REGION Network 4: Current revision and modification history
   // ▄▄▄▄▄▄▄▄▄▄▄▄▄▄▄▄▄▄▄▄▄▄▄▄▄▄▄▄▄▄▄▄▄▄▄▄▄▄▄▄▄▄▄▄
   // MODIFICATION HISTORY
   // 
   // 
   // The revision data shown here, in the network comments, contains additional information 
   // reflecting the software development workflow under the version control system (VCS) employed 
   // to track all software changes.
   // 
   // The VCS in use is the Git Source Code Management system in conjunction with the GitHub online 
   // hosting system. The software in its entirety is available in the GitHub remote repository:
   // 
   //      https://github.com/practicalseries/PS2001-pal-software
   // 
   // The repository is public and can be freely copied (forked in GitHub terminology) and used 
   // under the MIT licence. 
   // 
   // The MIT licence is reproduced in full in the last network of this software module.
   // 
   // 
   //  ―――――――――――――――――――――――――――――――――――――――――――
   //  DATE       REVISION             MASTER BRANCH     DEV
   //          (nnn.amm)   COMMIT TAG    (Base ---> Merge)    BRANCH   Author
   //  ———————————————————————————————————————————
   //  2024.05.11    002.801   D0017A-000.104   D0017 N/A     D017A   M. Gledhill
   //                        RAW_ANALOG changed to AI_RAW_SIGNAL
   //                        AI_RAW_DATA and AI_SCALE_DATA added and
   //                        copied to DYNAMIC_DATA (see db00801 SMDS)
   // 
   //  2022.04.16    002.000   D0011      D0010 D0011  None  M. Gledhill
   //                        FC02001 — RELEASED FOR USE
   //                          Merge back to master branch
   // 
   //  2022.04.11    001.801   D0010A-000.801   D0010 N/A     D010A   M. Gledhill
   //                        Released for test (SCV)
   //  2022.04.08    001.102   D0010A-000.104   D0010 N/A     D010A   M. Gledhill
   //                        Temporary variable name change (cal)
   // 
   //  2022.04.05    001.101   D0010A-000.103   D0010 N/A     D010A   M. Gledhill
   //                        Over and under range based on scaled signal
   //                        INFO_TYPE, cal_OR_Abs and cal_UR_Abs added
   //                        Comments updated and standardised
   //                        UDT variable names standardised
   // 
   //  2021.05.26    001.000   D0008      D0006 D0008  None    M. Gledhill
   //                        FC02001 — RELEASED FOR USE
   //                          Merge back to master branch
   // 
   //  2021.05.26    001.000   D0006B-001.000   D0006 N/A     D0006B   M. Gledhill
   //                        FC02001 — Post-test RELEASED FOR USE
   // 
   //  2021.05.24    000.801   D0006B-000.801   D0006 N/A     D0006B   M. Gledhill
   //                        FC02001 — Released for SMT
   // 
   //  2021.05.18    000.101   D0006B-000.101   D0006 N/A     D0006B   M. Gledhill
   //                        FC02001 Migration to VCS
   //  ———————————————————————————————————————————
   //   Where: nnn  =  Major revision
   //         a  =  Type (1-7 Development, 8 Proving, 9 Qualification, 0 Release)
   //       mm  =  Minor revision (must be 00 if a = 0)
   //         Block properties version number should be set to nn.a (only one decimal place)
   // 
   // ▄▄▄▄▄▄▄▄▄▄▄▄▄▄▄▄▄▄▄▄▄▄▄▄▄▄▄▄▄▄▄▄▄▄▄▄▄▄▄▄▄▄▄▄
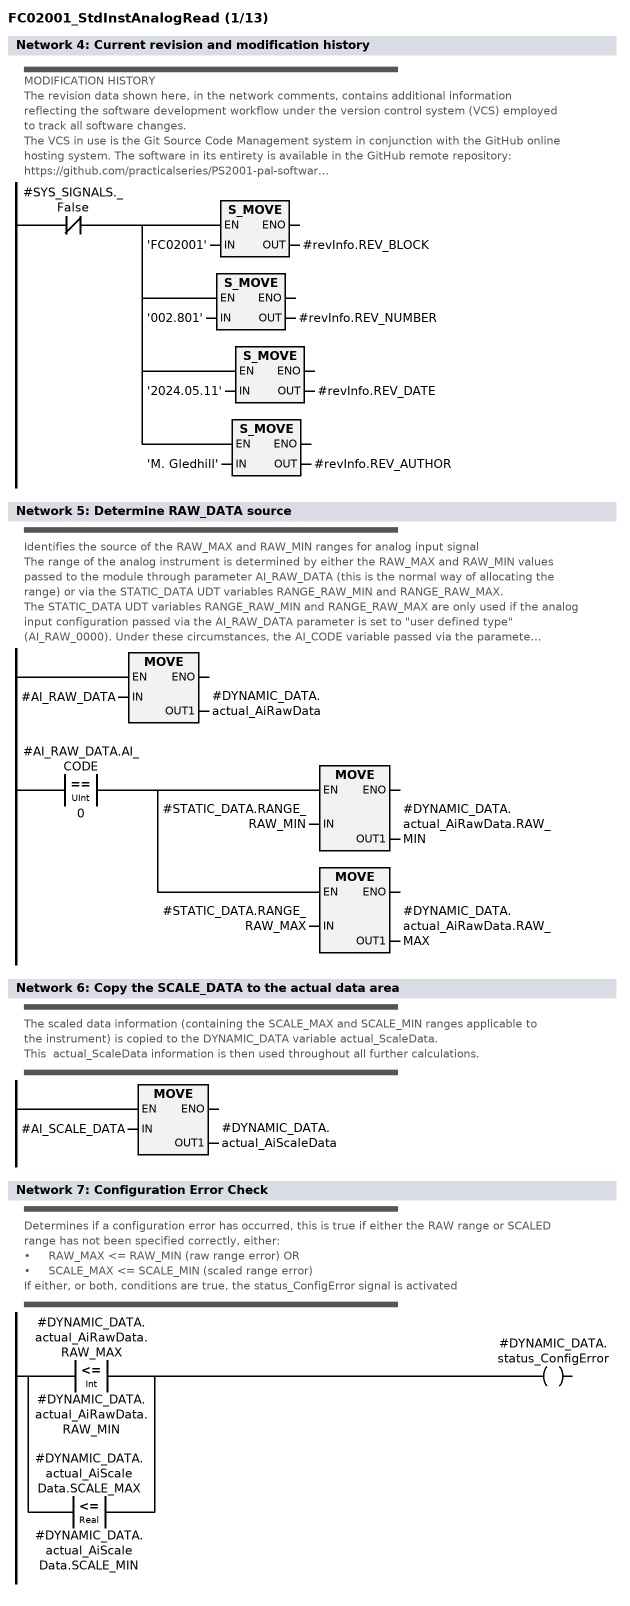
   RUNG wire#powerrail
      I_Contact( #SYS_SIGNALS._False )
      wire#w1
      S_Move(in := 'FC02001', out => #revInfo.REV_BLOCK)
   END_RUNG
   RUNG wire#w1
      S_Move(in := '002.801', out => #revInfo.REV_NUMBER)
   END_RUNG
   RUNG wire#w1
      S_Move(in := '2024.05.11', out => #revInfo.REV_DATE)
   END_RUNG
   RUNG wire#w1
      S_Move(in := 'M. Gledhill', out => #revInfo.REV_AUTHOR)
   END_RUNG
   // the same network as SCL:
   IF NOT #SYS_SIGNALS._False THEN
       #revInfo.REV_BLOCK := 'FC02001';
       #revInfo.REV_NUMBER := '002.801';
       #revInfo.REV_DATE := '2024.05.11';
       #revInfo.REV_AUTHOR := 'M. Gledhill';
   END_IF;
END_REGION

REGION Network 5: Determine RAW_DATA source
   // ▀▀▀▀▀▀▀▀▀▀▀▀▀▀▀▀▀▀▀▀▀▀▀▀▀▀▀▀▀▀▀▀▀▀▀▀▀▀▀▀▀▀▀▀
   // Identifies the source of the RAW_MAX and RAW_MIN ranges for analog input signal
   // 
   // The range of the analog instrument is determined by either the RAW_MAX and RAW_MIN values 
   // passed to the module through parameter AI_RAW_DATA (this is the normal way of allocating the 
   // range) or via the STATIC_DATA UDT variables RANGE_RAW_MIN and RANGE_RAW_MAX.
   // 
   // 
   // The STATIC_DATA UDT variables RANGE_RAW_MIN and RANGE_RAW_MAX are only used if the analog
   // input configuration passed via the AI_RAW_DATA parameter is set to "user defined type" 
   // (AI_RAW_0000). Under these circumstances, the AI_CODE variable passed via the parameter 
   // AI_RAW_DATA will be set to zero and the STATIC_DATA UDT variables RANGE_RAW_MIN and 
   // RANGE_RAW_MAX are to be used in place of the range data given via the AI_RAW_DATA parameter.
   // 
   // Irrespective of the source, the RAW_MIN and RAW_MAX data in use will be copied to the 
   // DYNAMIC_DATA variable actual_RawData.
   // ▄▄▄▄▄▄▄▄▄▄▄▄▄▄▄▄▄▄▄▄▄▄▄▄▄▄▄▄▄▄▄▄▄▄▄▄▄▄▄▄▄▄▄▄
   RUNG wire#powerrail
      Move(in := #AI_RAW_DATA, out1 => #DYNAMIC_DATA.actual_AiRawData)
   END_RUNG
   RUNG wire#powerrail
      { S7_Templates := "SrcType := UInt" } EQ_Contact(in1 := #AI_RAW_DATA.AI_CODE, in2 := 0)
      wire#w1
      Move(in := #STATIC_DATA.RANGE_RAW_MIN, out1 => #DYNAMIC_DATA.actual_AiRawData.RAW_MIN)
   END_RUNG
   RUNG wire#w1
      Move(in := #STATIC_DATA.RANGE_RAW_MAX, out1 => #DYNAMIC_DATA.actual_AiRawData.RAW_MAX)
   END_RUNG
   // the same network as SCL:
   #DYNAMIC_DATA.actual_AiRawData := #AI_RAW_DATA;
   IF #AI_RAW_DATA.AI_CODE = 0 THEN
       #DYNAMIC_DATA.actual_AiRawData.RAW_MIN := #STATIC_DATA.RANGE_RAW_MIN;
       #DYNAMIC_DATA.actual_AiRawData.RAW_MAX := #STATIC_DATA.RANGE_RAW_MAX;
   END_IF;
END_REGION

REGION Network 6: Copy the SCALE_DATA to the actual data area
   // ▀▀▀▀▀▀▀▀▀▀▀▀▀▀▀▀▀▀▀▀▀▀▀▀▀▀▀▀▀▀▀▀▀▀▀▀▀▀▀▀▀▀▀▀
   // The scaled data information (containing the SCALE_MAX and SCALE_MIN ranges applicable to
   // the instrument) is copied to the DYNAMIC_DATA variable actual_ScaleData.
   // 
   // This  actual_ScaleData information is then used throughout all further calculations.
   // ▄▄▄▄▄▄▄▄▄▄▄▄▄▄▄▄▄▄▄▄▄▄▄▄▄▄▄▄▄▄▄▄▄▄▄▄▄▄▄▄▄▄▄▄
   RUNG wire#powerrail
      Move(in := #AI_SCALE_DATA, out1 => #DYNAMIC_DATA.actual_AiScaleData)
   END_RUNG
   // the same network as SCL:
   #DYNAMIC_DATA.actual_AiScaleData := #AI_SCALE_DATA;
END_REGION

REGION Network 7: Configuration Error Check
   // ▀▀▀▀▀▀▀▀▀▀▀▀▀▀▀▀▀▀▀▀▀▀▀▀▀▀▀▀▀▀▀▀▀▀▀▀▀▀▀▀▀▀▀▀
   // Determines if a configuration error has occurred, this is true if either the RAW range or SCALED 
   // range has not been specified correctly, either:
   // 
   //    •   RAW_MAX <= RAW_MIN (raw range error) OR
   //    •   SCALE_MAX <= SCALE_MIN (scaled range error)
   // 
   // If either, or both, conditions are true, the status_ConfigError signal is activated
   // ▄▄▄▄▄▄▄▄▄▄▄▄▄▄▄▄▄▄▄▄▄▄▄▄▄▄▄▄▄▄▄▄▄▄▄▄▄▄▄▄▄▄▄▄
   RUNG wire#powerrail
      { S7_Templates := "SrcType := Int" } LE_Contact(in1 := #DYNAMIC_DATA.actual_AiRawData.RAW_MAX, in2 := #DYNAMIC_DATA.actual_AiRawData.RAW_MIN)
      wire#w1
      Coil( #DYNAMIC_DATA.status_ConfigError )
   END_RUNG
   RUNG wire#powerrail
      { S7_Templates := "SrcType := Real" } LE_Contact(in1 := #DYNAMIC_DATA.actual_AiScaleData.SCALE_MAX, in2 := #DYNAMIC_DATA.actual_AiScaleData.SCALE_MIN)
   END_RUNG wire#w1
   // the same network as SCL:
   #DYNAMIC_DATA.status_ConfigError := (#DYNAMIC_DATA.actual_AiRawData.RAW_MAX <= #DYNAMIC_DATA.actual_AiRawData.RAW_MIN) OR (#DYNAMIC_DATA.actual_AiScaleData.SCALE_MAX <= #DYNAMIC_DATA.actual_AiScaleData.SCALE_MIN);
END_REGION

REGION Network 8: Signal Conditioning — Simulation mode disabled
   // ▀▀▀▀▀▀▀▀▀▀▀▀▀▀▀▀▀▀▀▀▀▀▀▀▀▀▀▀▀▀▀▀▀▀▀▀▀▀▀▀▀▀▀▀
   // If simulation mode is disabled (CONFIG_SIM_DIS = 1), or if the faceplate is disabled 
   // (CONFIG_FP_DIS = 1),reset any simulation mode activation signal.
   // ▄▄▄▄▄▄▄▄▄▄▄▄▄▄▄▄▄▄▄▄▄▄▄▄▄▄▄▄▄▄▄▄▄▄▄▄▄▄▄▄▄▄▄▄
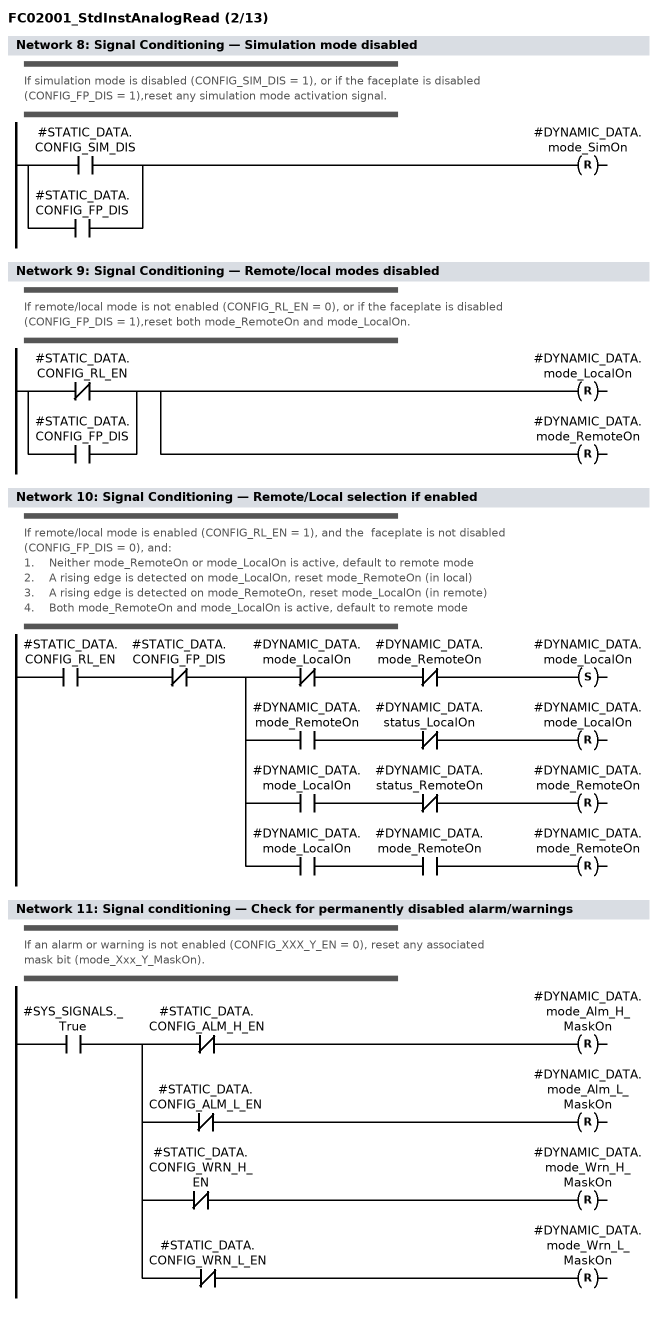
   RUNG wire#powerrail
      Contact( #STATIC_DATA.CONFIG_SIM_DIS )
      wire#w1
      R_Coil( #DYNAMIC_DATA.mode_SimOn )
   END_RUNG
   RUNG wire#powerrail
      Contact( #STATIC_DATA.CONFIG_FP_DIS )
   END_RUNG wire#w1
   // the same network as SCL:
   IF #STATIC_DATA.CONFIG_SIM_DIS OR #STATIC_DATA.CONFIG_FP_DIS THEN
       #DYNAMIC_DATA.mode_SimOn := FALSE;
   END_IF;
END_REGION

REGION Network 9: Signal Conditioning — Remote/local modes disabled
   // ▀▀▀▀▀▀▀▀▀▀▀▀▀▀▀▀▀▀▀▀▀▀▀▀▀▀▀▀▀▀▀▀▀▀▀▀▀▀▀▀▀▀▀▀
   // If remote/local mode is not enabled (CONFIG_RL_EN = 0), or if the faceplate is disabled 
   // (CONFIG_FP_DIS = 1),reset both mode_RemoteOn and mode_LocalOn.
   // ▄▄▄▄▄▄▄▄▄▄▄▄▄▄▄▄▄▄▄▄▄▄▄▄▄▄▄▄▄▄▄▄▄▄▄▄▄▄▄▄▄▄▄▄
   RUNG wire#powerrail
      I_Contact( #STATIC_DATA.CONFIG_RL_EN )
      wire#w1
      R_Coil( #DYNAMIC_DATA.mode_LocalOn )
   END_RUNG
   RUNG wire#powerrail
      Contact( #STATIC_DATA.CONFIG_FP_DIS )
   END_RUNG wire#w1
   RUNG wire#w1
      R_Coil( #DYNAMIC_DATA.mode_RemoteOn )
   END_RUNG
   // the same network as SCL:
   IF NOT #STATIC_DATA.CONFIG_RL_EN OR #STATIC_DATA.CONFIG_FP_DIS THEN
       #DYNAMIC_DATA.mode_LocalOn := FALSE;
       #DYNAMIC_DATA.mode_RemoteOn := FALSE;
   END_IF;
END_REGION

REGION Network 10: Signal Conditioning — Remote/Local selection if enabled
   // ▀▀▀▀▀▀▀▀▀▀▀▀▀▀▀▀▀▀▀▀▀▀▀▀▀▀▀▀▀▀▀▀▀▀▀▀▀▀▀▀▀▀▀▀
   // If remote/local mode is enabled (CONFIG_RL_EN = 1), and the  faceplate is not disabled 
   // (CONFIG_FP_DIS = 0), and:
   // 
   //    1.  Neither mode_RemoteOn or mode_LocalOn is active, default to remote mode
   //    2.  A rising edge is detected on mode_LocalOn, reset mode_RemoteOn (in local)
   //    3.  A rising edge is detected on mode_RemoteOn, reset mode_LocalOn (in remote)
   //    4.  Both mode_RemoteOn and mode_LocalOn is active, default to remote mode
   // ▄▄▄▄▄▄▄▄▄▄▄▄▄▄▄▄▄▄▄▄▄▄▄▄▄▄▄▄▄▄▄▄▄▄▄▄▄▄▄▄▄▄▄▄
   RUNG wire#powerrail
      Contact( #STATIC_DATA.CONFIG_RL_EN )
      I_Contact( #STATIC_DATA.CONFIG_FP_DIS )
      wire#w1
      I_Contact( #DYNAMIC_DATA.mode_LocalOn )
      I_Contact( #DYNAMIC_DATA.mode_RemoteOn )
      S_Coil( #DYNAMIC_DATA.mode_LocalOn )
   END_RUNG
   RUNG wire#w1
      Contact( #DYNAMIC_DATA.mode_RemoteOn )
      I_Contact( #DYNAMIC_DATA.status_LocalOn )
      R_Coil( #DYNAMIC_DATA.mode_LocalOn )
   END_RUNG
   RUNG wire#w1
      Contact( #DYNAMIC_DATA.mode_LocalOn )
      I_Contact( #DYNAMIC_DATA.status_RemoteOn )
      R_Coil( #DYNAMIC_DATA.mode_RemoteOn )
   END_RUNG
   RUNG wire#w1
      Contact( #DYNAMIC_DATA.mode_LocalOn )
      Contact( #DYNAMIC_DATA.mode_RemoteOn )
      R_Coil( #DYNAMIC_DATA.mode_RemoteOn )
   END_RUNG
   // the same network as SCL:
   #_w1 := #STATIC_DATA.CONFIG_RL_EN AND NOT #STATIC_DATA.CONFIG_FP_DIS;
   IF #_w1 AND NOT #DYNAMIC_DATA.mode_LocalOn AND NOT #DYNAMIC_DATA.mode_RemoteOn THEN
       #DYNAMIC_DATA.mode_LocalOn := TRUE;
   END_IF;
   IF #_w1 AND #DYNAMIC_DATA.mode_RemoteOn AND NOT #DYNAMIC_DATA.status_LocalOn THEN
       #DYNAMIC_DATA.mode_LocalOn := FALSE;
   END_IF;
   IF #_w1 AND #DYNAMIC_DATA.mode_LocalOn AND NOT #DYNAMIC_DATA.status_RemoteOn THEN
       #DYNAMIC_DATA.mode_RemoteOn := FALSE;
   END_IF;
   IF #_w1 AND #DYNAMIC_DATA.mode_LocalOn AND #DYNAMIC_DATA.mode_RemoteOn THEN
       #DYNAMIC_DATA.mode_RemoteOn := FALSE;
   END_IF;
END_REGION

REGION Network 11: Signal conditioning — Check for permanently disabled alarm/warnings
   // ▀▀▀▀▀▀▀▀▀▀▀▀▀▀▀▀▀▀▀▀▀▀▀▀▀▀▀▀▀▀▀▀▀▀▀▀▀▀▀▀▀▀▀▀
   // If an alarm or warning is not enabled (CONFIG_XXX_Y_EN = 0), reset any associated 
   // mask bit (mode_Xxx_Y_MaskOn).
   // ▄▄▄▄▄▄▄▄▄▄▄▄▄▄▄▄▄▄▄▄▄▄▄▄▄▄▄▄▄▄▄▄▄▄▄▄▄▄▄▄▄▄▄▄
   RUNG wire#powerrail
      Contact( #SYS_SIGNALS._True )
      wire#w1
      I_Contact( #STATIC_DATA.CONFIG_ALM_H_EN )
      R_Coil( #DYNAMIC_DATA.mode_Alm_H_MaskOn )
   END_RUNG
   RUNG wire#w1
      I_Contact( #STATIC_DATA.CONFIG_ALM_L_EN )
      R_Coil( #DYNAMIC_DATA.mode_Alm_L_MaskOn )
   END_RUNG
   RUNG wire#w1
      I_Contact( #STATIC_DATA.CONFIG_WRN_H_EN )
      R_Coil( #DYNAMIC_DATA.mode_Wrn_H_MaskOn )
   END_RUNG
   RUNG wire#w1
      I_Contact( #STATIC_DATA.CONFIG_WRN_L_EN )
      R_Coil( #DYNAMIC_DATA.mode_Wrn_L_MaskOn )
   END_RUNG
   // the same network as SCL:
   IF #SYS_SIGNALS._True AND NOT #STATIC_DATA.CONFIG_ALM_H_EN THEN
       #DYNAMIC_DATA.mode_Alm_H_MaskOn := FALSE;
   END_IF;
   IF #SYS_SIGNALS._True AND NOT #STATIC_DATA.CONFIG_ALM_L_EN THEN
       #DYNAMIC_DATA.mode_Alm_L_MaskOn := FALSE;
   END_IF;
   IF #SYS_SIGNALS._True AND NOT #STATIC_DATA.CONFIG_WRN_H_EN THEN
       #DYNAMIC_DATA.mode_Wrn_H_MaskOn := FALSE;
   END_IF;
   IF #SYS_SIGNALS._True AND NOT #STATIC_DATA.CONFIG_WRN_L_EN THEN
       #DYNAMIC_DATA.mode_Wrn_L_MaskOn := FALSE;
   END_IF;
END_REGION

REGION Network 12: Signal conditioning — Identify alarm/warnings that are to be evaluated
   // ▀▀▀▀▀▀▀▀▀▀▀▀▀▀▀▀▀▀▀▀▀▀▀▀▀▀▀▀▀▀▀▀▀▀▀▀▀▀▀▀▀▀▀▀
   // If an alarm or warning is both ENABLED and NOT MASKED then the associated (local data) 
   // working bit wrkXxxYEn bit is set; this is used in the following networks to indicate that the 
   // alarm/warning is to be evaluated.
   // ▄▄▄▄▄▄▄▄▄▄▄▄▄▄▄▄▄▄▄▄▄▄▄▄▄▄▄▄▄▄▄▄▄▄▄▄▄▄▄▄▄▄▄▄
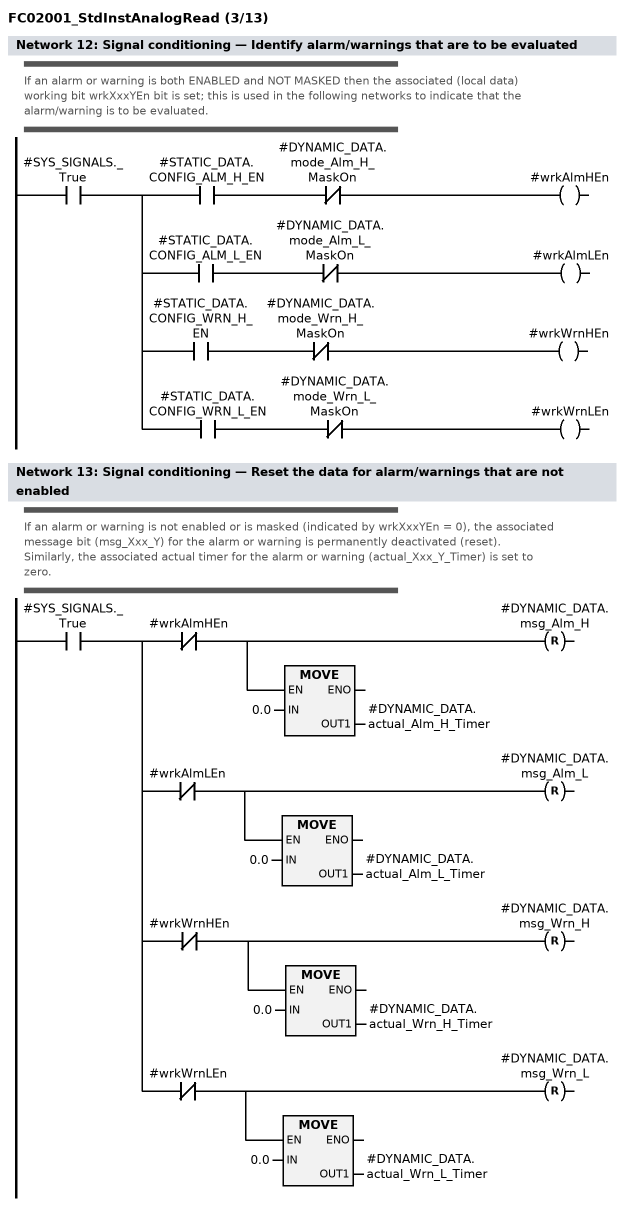
   RUNG wire#powerrail
      Contact( #SYS_SIGNALS._True )
      wire#w1
      Contact( #STATIC_DATA.CONFIG_ALM_H_EN )
      I_Contact( #DYNAMIC_DATA.mode_Alm_H_MaskOn )
      Coil( #wrkAlmHEn )
   END_RUNG
   RUNG wire#w1
      Contact( #STATIC_DATA.CONFIG_ALM_L_EN )
      I_Contact( #DYNAMIC_DATA.mode_Alm_L_MaskOn )
      Coil( #wrkAlmLEn )
   END_RUNG
   RUNG wire#w1
      Contact( #STATIC_DATA.CONFIG_WRN_H_EN )
      I_Contact( #DYNAMIC_DATA.mode_Wrn_H_MaskOn )
      Coil( #wrkWrnHEn )
   END_RUNG
   RUNG wire#w1
      Contact( #STATIC_DATA.CONFIG_WRN_L_EN )
      I_Contact( #DYNAMIC_DATA.mode_Wrn_L_MaskOn )
      Coil( #wrkWrnLEn )
   END_RUNG
   // the same network as SCL:
   #wrkAlmHEn := #SYS_SIGNALS._True AND #STATIC_DATA.CONFIG_ALM_H_EN AND NOT #DYNAMIC_DATA.mode_Alm_H_MaskOn;
   #wrkAlmLEn := #SYS_SIGNALS._True AND #STATIC_DATA.CONFIG_ALM_L_EN AND NOT #DYNAMIC_DATA.mode_Alm_L_MaskOn;
   #wrkWrnHEn := #SYS_SIGNALS._True AND #STATIC_DATA.CONFIG_WRN_H_EN AND NOT #DYNAMIC_DATA.mode_Wrn_H_MaskOn;
   #wrkWrnLEn := #SYS_SIGNALS._True AND #STATIC_DATA.CONFIG_WRN_L_EN AND NOT #DYNAMIC_DATA.mode_Wrn_L_MaskOn;
END_REGION

REGION Network 13: Signal conditioning — Reset the data for alarm/warnings that are not enabled
   // ▀▀▀▀▀▀▀▀▀▀▀▀▀▀▀▀▀▀▀▀▀▀▀▀▀▀▀▀▀▀▀▀▀▀▀▀▀▀▀▀▀▀▀▀
   // If an alarm or warning is not enabled or is masked (indicated by wrkXxxYEn = 0), the associated 
   // message bit (msg_Xxx_Y) for the alarm or warning is permanently deactivated (reset).
   // 
   // Similarly, the associated actual timer for the alarm or warning (actual_Xxx_Y_Timer) is set to 
   // zero.
   // ▄▄▄▄▄▄▄▄▄▄▄▄▄▄▄▄▄▄▄▄▄▄▄▄▄▄▄▄▄▄▄▄▄▄▄▄▄▄▄▄▄▄▄▄
   RUNG wire#powerrail
      Contact( #SYS_SIGNALS._True )
      wire#w1
      I_Contact( #wrkAlmHEn )
      wire#w2
      R_Coil( #DYNAMIC_DATA.msg_Alm_H )
   END_RUNG
   RUNG wire#w2
      { S7_GenerateENO := "TRUE" } Move(in := 0.0, out1 => #DYNAMIC_DATA.actual_Alm_H_Timer)
   END_RUNG
   RUNG wire#w1
      I_Contact( #wrkAlmLEn )
      wire#w3
      R_Coil( #DYNAMIC_DATA.msg_Alm_L )
   END_RUNG
   RUNG wire#w3
      { S7_GenerateENO := "TRUE" } Move(in := 0.0, out1 => #DYNAMIC_DATA.actual_Alm_L_Timer)
   END_RUNG
   RUNG wire#w1
      I_Contact( #wrkWrnHEn )
      wire#w4
      R_Coil( #DYNAMIC_DATA.msg_Wrn_H )
   END_RUNG
   RUNG wire#w4
      { S7_GenerateENO := "TRUE" } Move(in := 0.0, out1 => #DYNAMIC_DATA.actual_Wrn_H_Timer)
   END_RUNG
   RUNG wire#w1
      I_Contact( #wrkWrnLEn )
      wire#w5
      R_Coil( #DYNAMIC_DATA.msg_Wrn_L )
   END_RUNG
   RUNG wire#w5
      { S7_GenerateENO := "TRUE" } Move(in := 0.0, out1 => #DYNAMIC_DATA.actual_Wrn_L_Timer)
   END_RUNG
   // the same network as SCL:
   IF #SYS_SIGNALS._True AND NOT #wrkAlmHEn THEN
       #DYNAMIC_DATA.msg_Alm_H := FALSE;
       #DYNAMIC_DATA.actual_Alm_H_Timer := 0.0;
   END_IF;
   IF #SYS_SIGNALS._True AND NOT #wrkAlmLEn THEN
       #DYNAMIC_DATA.msg_Alm_L := FALSE;
       #DYNAMIC_DATA.actual_Alm_L_Timer := 0.0;
   END_IF;
   IF #SYS_SIGNALS._True AND NOT #wrkWrnHEn THEN
       #DYNAMIC_DATA.msg_Wrn_H := FALSE;
       #DYNAMIC_DATA.actual_Wrn_H_Timer := 0.0;
   END_IF;
   IF #SYS_SIGNALS._True AND NOT #wrkWrnLEn THEN
       #DYNAMIC_DATA.msg_Wrn_L := FALSE;
       #DYNAMIC_DATA.actual_Wrn_L_Timer := 0.0;
   END_IF;
END_REGION

REGION Network 14: Signal conditioning — Detect recently enabled alarm/warnings
   // ▀▀▀▀▀▀▀▀▀▀▀▀▀▀▀▀▀▀▀▀▀▀▀▀▀▀▀▀▀▀▀▀▀▀▀▀▀▀▀▀▀▀▀▀
   // If the working alarm or warning enable signal (wrkXxxYEn) changes to a high state
   // (i.e. the alarm is enabled during run-time), the alarm/warning timer (actual_Xxx_Y_Timer) is 
   // pre-loaded with the ON-DELAY time (TIME_XXX_Y_ON_DEL).
   // 
   // This prevents the alarm/warning from activating instantly, if the actual_Value is outside the
   // alarm/warning setpoint. This condition could arise because the timer is set to zero while ever
   // the alarm/warning is disabled.
   // 
   // Note:    Technically, the ENABLE bit should not be modified at run-time, it is stored in a static
   //      data block; however, the condition could arise if that static data block is being used
   //      as a recipe block. mask signals can of course be changed at run-time.
   // ▄▄▄▄▄▄▄▄▄▄▄▄▄▄▄▄▄▄▄▄▄▄▄▄▄▄▄▄▄▄▄▄▄▄▄▄▄▄▄▄▄▄▄▄
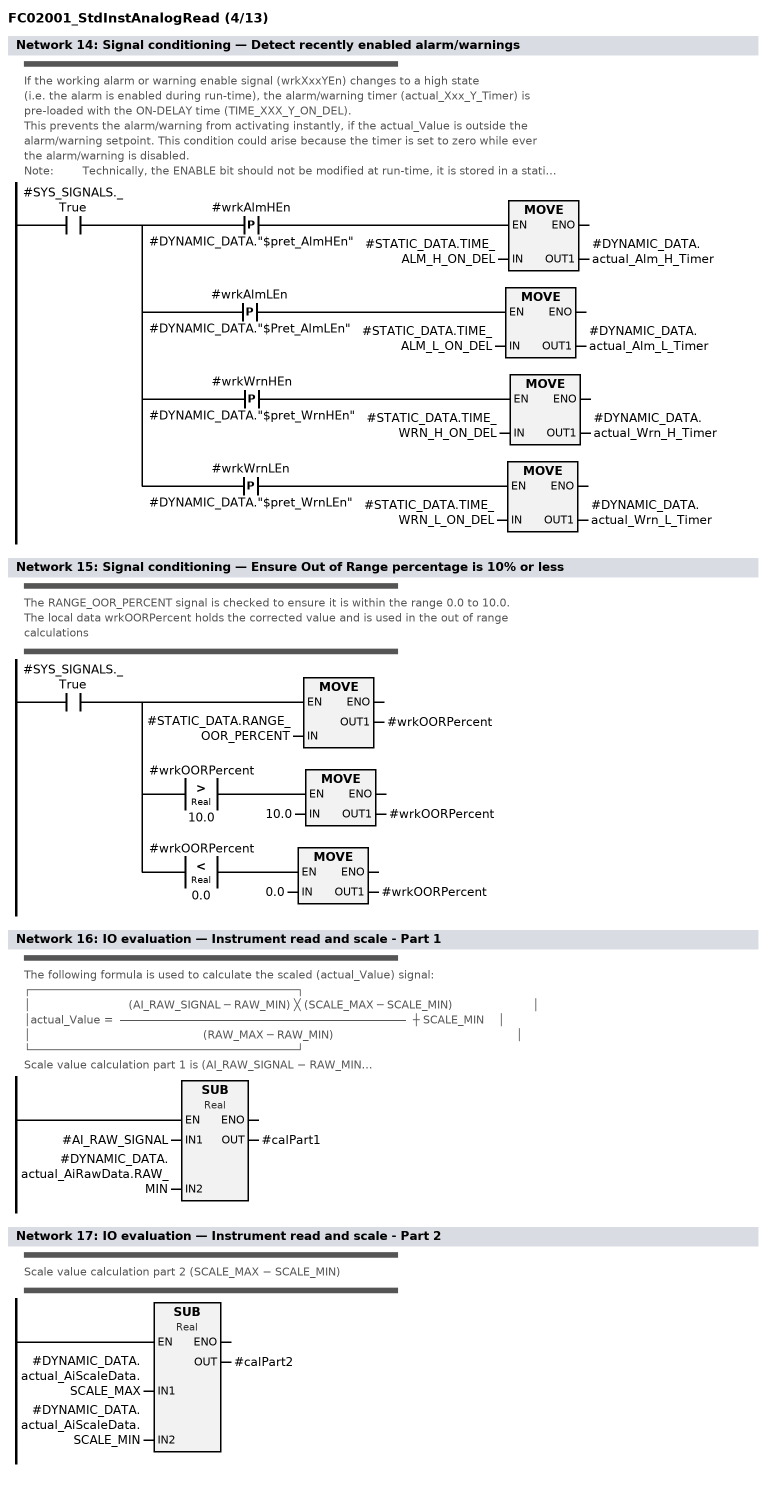
   RUNG wire#powerrail
      Contact( #SYS_SIGNALS._True )
      wire#w1
      P_Contact(operand := #wrkAlmHEn, bit := #DYNAMIC_DATA."$pret_AlmHEn")
      { S7_GenerateENO := "TRUE" } Move(in := #STATIC_DATA.TIME_ALM_H_ON_DEL, out1 => #DYNAMIC_DATA.actual_Alm_H_Timer)
   END_RUNG
   RUNG wire#w1
      P_Contact(operand := #wrkAlmLEn, bit := #DYNAMIC_DATA."$Pret_AlmLEn")
      { S7_GenerateENO := "TRUE" } Move(in := #STATIC_DATA.TIME_ALM_L_ON_DEL, out1 => #DYNAMIC_DATA.actual_Alm_L_Timer)
   END_RUNG
   RUNG wire#w1
      P_Contact(operand := #wrkWrnHEn, bit := #DYNAMIC_DATA."$pret_WrnHEn")
      { S7_GenerateENO := "TRUE" } Move(in := #STATIC_DATA.TIME_WRN_H_ON_DEL, out1 => #DYNAMIC_DATA.actual_Wrn_H_Timer)
   END_RUNG
   RUNG wire#w1
      P_Contact(operand := #wrkWrnLEn, bit := #DYNAMIC_DATA."$pret_WrnLEn")
      { S7_GenerateENO := "TRUE" } Move(in := #STATIC_DATA.TIME_WRN_L_ON_DEL, out1 => #DYNAMIC_DATA.actual_Wrn_L_Timer)
   END_RUNG
   // the same network as SCL:
   #_w1 := #SYS_SIGNALS._True AND #wrkAlmHEn AND NOT #DYNAMIC_DATA."$pret_AlmHEn";   // rising edge of #wrkAlmHEn
   #DYNAMIC_DATA."$pret_AlmHEn" := #wrkAlmHEn;
   IF #_w1 THEN #DYNAMIC_DATA.actual_Alm_H_Timer := #STATIC_DATA.TIME_ALM_H_ON_DEL; END_IF;
   #_w2 := #SYS_SIGNALS._True AND #wrkAlmLEn AND NOT #DYNAMIC_DATA."$Pret_AlmLEn";   // rising edge of #wrkAlmLEn
   #DYNAMIC_DATA."$Pret_AlmLEn" := #wrkAlmLEn;
   IF #_w2 THEN #DYNAMIC_DATA.actual_Alm_L_Timer := #STATIC_DATA.TIME_ALM_L_ON_DEL; END_IF;
   #_w3 := #SYS_SIGNALS._True AND #wrkWrnHEn AND NOT #DYNAMIC_DATA."$pret_WrnHEn";   // rising edge of #wrkWrnHEn
   #DYNAMIC_DATA."$pret_WrnHEn" := #wrkWrnHEn;
   IF #_w3 THEN #DYNAMIC_DATA.actual_Wrn_H_Timer := #STATIC_DATA.TIME_WRN_H_ON_DEL; END_IF;
   #_w4 := #SYS_SIGNALS._True AND #wrkWrnLEn AND NOT #DYNAMIC_DATA."$pret_WrnLEn";   // rising edge of #wrkWrnLEn
   #DYNAMIC_DATA."$pret_WrnLEn" := #wrkWrnLEn;
   IF #_w4 THEN #DYNAMIC_DATA.actual_Wrn_L_Timer := #STATIC_DATA.TIME_WRN_L_ON_DEL; END_IF;
END_REGION

REGION Network 15: Signal conditioning — Ensure Out of Range percentage is 10% or less
   // ▀▀▀▀▀▀▀▀▀▀▀▀▀▀▀▀▀▀▀▀▀▀▀▀▀▀▀▀▀▀▀▀▀▀▀▀▀▀▀▀▀▀▀▀
   // The RANGE_OOR_PERCENT signal is checked to ensure it is within the range 0.0 to 10.0.
   // 
   // The local data wrkOORPercent holds the corrected value and is used in the out of range 
   // calculations
   // ▄▄▄▄▄▄▄▄▄▄▄▄▄▄▄▄▄▄▄▄▄▄▄▄▄▄▄▄▄▄▄▄▄▄▄▄▄▄▄▄▄▄▄▄
   RUNG wire#powerrail
      Contact( #SYS_SIGNALS._True )
      wire#w1
      { S7_GenerateENO := "TRUE" } Move(in := #STATIC_DATA.RANGE_OOR_PERCENT, out1 => #wrkOORPercent)
   END_RUNG
   RUNG wire#w1
      { S7_Templates := "SrcType := Real" } GT_Contact(in1 := #wrkOORPercent, in2 := 10.0)
      { S7_GenerateENO := "TRUE" } Move(in := 10.0, out1 => #wrkOORPercent)
   END_RUNG
   RUNG wire#w1
      { S7_Templates := "SrcType := Real" } LT_Contact(in1 := #wrkOORPercent, in2 := 0.0)
      { S7_GenerateENO := "TRUE" } Move(in := 0.0, out1 => #wrkOORPercent)
   END_RUNG
   // the same network as SCL:
   IF #SYS_SIGNALS._True THEN #wrkOORPercent := #STATIC_DATA.RANGE_OOR_PERCENT; END_IF;
   IF #SYS_SIGNALS._True AND (#wrkOORPercent > 10.0) THEN #wrkOORPercent := 10.0; END_IF;
   IF #SYS_SIGNALS._True AND (#wrkOORPercent < 0.0) THEN #wrkOORPercent := 0.0; END_IF;
END_REGION

REGION Network 16: IO evaluation — Instrument read and scale - Part 1
   // ▀▀▀▀▀▀▀▀▀▀▀▀▀▀▀▀▀▀▀▀▀▀▀▀▀▀▀▀▀▀▀▀▀▀▀▀▀▀▀▀▀▀▀▀
   // The following formula is used to calculate the scaled (actual_Value) signal:
   // ┌─────────────────────────────────────────┐
   // │                            (AI_RAW_SIGNAL ─ RAW_MIN) ╳ (SCALE_MAX ─ SCALE_MIN)          │
   // │actual_Value =  ――――――――――――――――――――――――――  ┼ SCALE_MIN    │
   // │                              (RAW_MAX ─ RAW_MIN)                    │
   // └─────────────────────────────────────────┘
   // 
   // 
   // Scale value calculation part 1 is (AI_RAW_SIGNAL − RAW_MIN)
   // ▄▄▄▄▄▄▄▄▄▄▄▄▄▄▄▄▄▄▄▄▄▄▄▄▄▄▄▄▄▄▄▄▄▄▄▄▄▄▄▄▄▄▄▄
   RUNG wire#powerrail
      { S7_Templates := "SrcType := Real"; S7_GenerateENO := "TRUE" } Sub(in1 := #AI_RAW_SIGNAL, in2 := #DYNAMIC_DATA.actual_AiRawData.RAW_MIN, out => #calPart1)
   END_RUNG
   // the same network as SCL:
   #calPart1 := #AI_RAW_SIGNAL - #DYNAMIC_DATA.actual_AiRawData.RAW_MIN;
END_REGION

REGION Network 17: IO evaluation — Instrument read and scale - Part 2
   // ▀▀▀▀▀▀▀▀▀▀▀▀▀▀▀▀▀▀▀▀▀▀▀▀▀▀▀▀▀▀▀▀▀▀▀▀▀▀▀▀▀▀▀▀
   // Scale value calculation part 2 (SCALE_MAX − SCALE_MIN)
   // ▄▄▄▄▄▄▄▄▄▄▄▄▄▄▄▄▄▄▄▄▄▄▄▄▄▄▄▄▄▄▄▄▄▄▄▄▄▄▄▄▄▄▄▄
   RUNG wire#powerrail
      { S7_Templates := "SrcType := Real"; S7_GenerateENO := "TRUE" } Sub(in1 := #DYNAMIC_DATA.actual_AiScaleData.SCALE_MAX, in2 := #DYNAMIC_DATA.actual_AiScaleData.SCALE_MIN, out => #calPart2)
   END_RUNG
   // the same network as SCL:
   #calPart2 := #DYNAMIC_DATA.actual_AiScaleData.SCALE_MAX - #DYNAMIC_DATA.actual_AiScaleData.SCALE_MIN;
END_REGION

REGION Network 18: IO evaluation — Instrument read and scale - Part 3
   // ▀▀▀▀▀▀▀▀▀▀▀▀▀▀▀▀▀▀▀▀▀▀▀▀▀▀▀▀▀▀▀▀▀▀▀▀▀▀▀▀▀▀▀▀
   // Scale value calculation part 3 (RAW_MAX − RAW_MIN)
   // 
   // Note:    To prevent inconsistencies and divide by zero errors, if a configuration error is present
   //      (resulting from incorrect range data and indicated by status_ConfigError = TRUE), the
   //      denominator of the calculation (CalPart3) is set to 3.402823 × 1038 (i.e. a very large 
   //      number), the result of this is that the  actual_Value will equal RANGE_SCALE_MIN for 
   //      all permitted values of AI_RAW_SIGNAL.
   // ▄▄▄▄▄▄▄▄▄▄▄▄▄▄▄▄▄▄▄▄▄▄▄▄▄▄▄▄▄▄▄▄▄▄▄▄▄▄▄▄▄▄▄▄
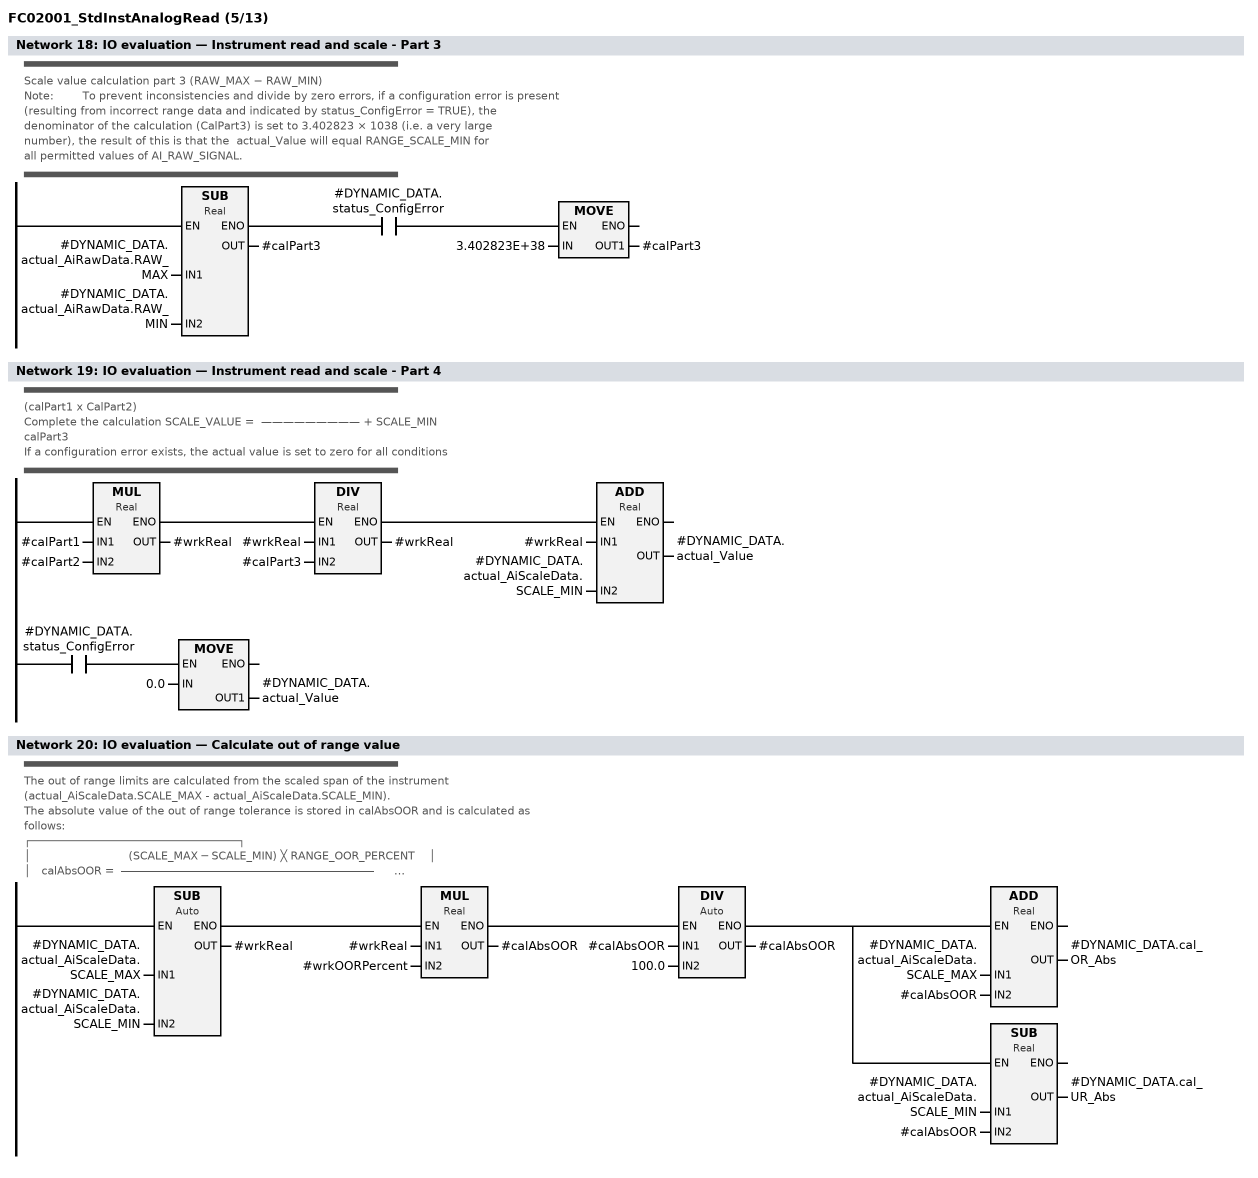
   RUNG wire#powerrail
      { S7_Templates := "SrcType := Real"; S7_GenerateENO := "TRUE" } Sub(in1 := #DYNAMIC_DATA.actual_AiRawData.RAW_MAX, in2 := #DYNAMIC_DATA.actual_AiRawData.RAW_MIN, out => #calPart3)
      Contact( #DYNAMIC_DATA.status_ConfigError )
      Move(in := 3.402823E+38, out1 => #calPart3)
   END_RUNG
   // the same network as SCL:
   // ENO of a box is taken as its EN; it also drops when the box reports an error
   #calPart3 := #DYNAMIC_DATA.actual_AiRawData.RAW_MAX - #DYNAMIC_DATA.actual_AiRawData.RAW_MIN;
   IF #DYNAMIC_DATA.status_ConfigError THEN #calPart3 := 3.402823E+38; END_IF;
END_REGION

REGION Network 19: IO evaluation — Instrument read and scale - Part 4
   // ▀▀▀▀▀▀▀▀▀▀▀▀▀▀▀▀▀▀▀▀▀▀▀▀▀▀▀▀▀▀▀▀▀▀▀▀▀▀▀▀▀▀▀▀
   //                                                                              (calPart1 x CalPart2)
   // Complete the calculation SCALE_VALUE =  ————————— + SCALE_MIN
   //                                                                                         calPart3
   // 
   // If a configuration error exists, the actual value is set to zero for all conditions
   // ▄▄▄▄▄▄▄▄▄▄▄▄▄▄▄▄▄▄▄▄▄▄▄▄▄▄▄▄▄▄▄▄▄▄▄▄▄▄▄▄▄▄▄▄
   RUNG wire#powerrail
      { S7_Templates := "SrcType := Real"; S7_GenerateENO := "TRUE" } Mul(in1 := #calPart1, in2 := #calPart2, out => #wrkReal)
      { S7_Templates := "SrcType := Real"; S7_GenerateENO := "TRUE" } Div(in1 := #wrkReal, in2 := #calPart3, out => #wrkReal)
      { S7_Templates := "SrcType := Real"; S7_GenerateENO := "TRUE" } Add(in1 := #wrkReal, in2 := #DYNAMIC_DATA.actual_AiScaleData.SCALE_MIN, out => #DYNAMIC_DATA.actual_Value)
   END_RUNG
   RUNG wire#powerrail
      Contact( #DYNAMIC_DATA.status_ConfigError )
      Move(in := 0.0, out1 => #DYNAMIC_DATA.actual_Value)
   END_RUNG
   // the same network as SCL:
   // ENO of a box is taken as its EN; it also drops when the box reports an error
   #wrkReal := #calPart1 * #calPart2;
   #wrkReal := #wrkReal / #calPart3;
   #DYNAMIC_DATA.actual_Value := #wrkReal + #DYNAMIC_DATA.actual_AiScaleData.SCALE_MIN;
   IF #DYNAMIC_DATA.status_ConfigError THEN #DYNAMIC_DATA.actual_Value := 0.0; END_IF;
END_REGION

REGION Network 20: IO evaluation — Calculate out of range value
   // ▀▀▀▀▀▀▀▀▀▀▀▀▀▀▀▀▀▀▀▀▀▀▀▀▀▀▀▀▀▀▀▀▀▀▀▀▀▀▀▀▀▀▀▀
   // The out of range limits are calculated from the scaled span of the instrument 
   // (actual_AiScaleData.SCALE_MAX - actual_AiScaleData.SCALE_MIN).
   // 
   // The absolute value of the out of range tolerance is stored in calAbsOOR and is calculated as
   // follows:
   // 
   // ┌────────────────────────────────┐
   // │                            (SCALE_MAX ─ SCALE_MIN) ╳ RANGE_OOR_PERCENT  │
   // │ calAbsOOR =  ―――――――――――――――――――――――    │
   // │                       100           │
   // └────────────────────────────────┘
   // 
   // The instrument is over range if the actual_Value is greater than SCALE_MAX + calcAbsOOR,
   // this absolute value is stored in the calculation variable cal_OR_Abs.
   // 
   // The instrument is under range if the AI_RAW_SIGNAL is less than SCALE_MIN - calcAbsOOR,
   // this absolute value is stored in the calculation variable cal_UR_Abs.
   // ▄▄▄▄▄▄▄▄▄▄▄▄▄▄▄▄▄▄▄▄▄▄▄▄▄▄▄▄▄▄▄▄▄▄▄▄▄▄▄▄▄▄▄▄
   RUNG wire#powerrail
      Sub(in1 := #DYNAMIC_DATA.actual_AiScaleData.SCALE_MAX, in2 := #DYNAMIC_DATA.actual_AiScaleData.SCALE_MIN, out => #wrkReal)
      { S7_Templates := "SrcType := Real"; S7_GenerateENO := "TRUE" } Mul(in1 := #wrkReal, in2 := #wrkOORPercent, out => #calAbsOOR)
      Div(in1 := #calAbsOOR, in2 := 100.0, out => #calAbsOOR)
      wire#w1
      { S7_Templates := "SrcType := Real"; S7_GenerateENO := "TRUE" } Add(in1 := #DYNAMIC_DATA.actual_AiScaleData.SCALE_MAX, in2 := #calAbsOOR, out => #DYNAMIC_DATA.cal_OR_Abs)
   END_RUNG
   RUNG wire#w1
      { S7_Templates := "SrcType := Real"; S7_GenerateENO := "TRUE" } Sub(in1 := #DYNAMIC_DATA.actual_AiScaleData.SCALE_MIN, in2 := #calAbsOOR, out => #DYNAMIC_DATA.cal_UR_Abs)
   END_RUNG
   // the same network as SCL:
   // ENO of a box is taken as its EN; it also drops when the box reports an error
   #wrkReal := #DYNAMIC_DATA.actual_AiScaleData.SCALE_MAX - #DYNAMIC_DATA.actual_AiScaleData.SCALE_MIN;
   #calAbsOOR := #wrkReal * #wrkOORPercent;
   #calAbsOOR := #calAbsOOR / 100.0;
   #DYNAMIC_DATA.cal_OR_Abs := #DYNAMIC_DATA.actual_AiScaleData.SCALE_MAX + #calAbsOOR;
   #DYNAMIC_DATA.cal_UR_Abs := #DYNAMIC_DATA.actual_AiScaleData.SCALE_MIN - #calAbsOOR;
END_REGION

REGION Network 21: IO evaluation — Out of range signals
   // ▀▀▀▀▀▀▀▀▀▀▀▀▀▀▀▀▀▀▀▀▀▀▀▀▀▀▀▀▀▀▀▀▀▀▀▀▀▀▀▀▀▀▀▀
   // The instrument is over range if the actual_Value is greater than or equal to cal_OR_Abs.
   // 
   // The instrument is under range if the actual_Value  is less than or equal to  cal_UR_Abs.
   // 
   // If either of these conditions is true, the common out of range signal is activated
   // 
   // Note:    The out of range signals are not generated if simulation mode is active
   // 
   // Note:    If the range information is incorrect (status_ConfigError = TRUE),
   //      Then all the out of range signals are activated msg_Flt_UnderRange, 
   //      msg_Flt_OverRange and msg_Flt_OutOfRange simultaneously, this is true even if
   //      simulation mode is active.
   // ▄▄▄▄▄▄▄▄▄▄▄▄▄▄▄▄▄▄▄▄▄▄▄▄▄▄▄▄▄▄▄▄▄▄▄▄▄▄▄▄▄▄▄▄
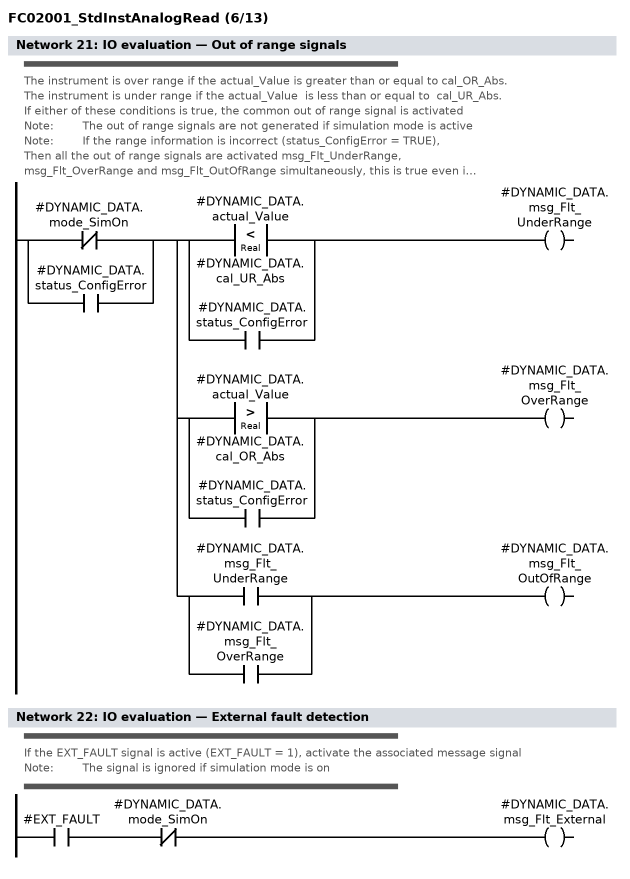
   RUNG wire#powerrail
      I_Contact( #DYNAMIC_DATA.mode_SimOn )
      wire#w1
      { S7_Templates := "SrcType := Real" } LT_Contact(in1 := #DYNAMIC_DATA.actual_Value, in2 := #DYNAMIC_DATA.cal_UR_Abs)
      wire#w2
      Coil( #DYNAMIC_DATA.msg_Flt_UnderRange )
   END_RUNG
   RUNG wire#powerrail
      Contact( #DYNAMIC_DATA.status_ConfigError )
   END_RUNG wire#w1
   RUNG wire#w1
      Contact( #DYNAMIC_DATA.status_ConfigError )
   END_RUNG wire#w2
   RUNG wire#w1
      { S7_Templates := "SrcType := Real" } GT_Contact(in1 := #DYNAMIC_DATA.actual_Value, in2 := #DYNAMIC_DATA.cal_OR_Abs)
      wire#w3
      Coil( #DYNAMIC_DATA.msg_Flt_OverRange )
   END_RUNG
   RUNG wire#w1
      Contact( #DYNAMIC_DATA.status_ConfigError )
   END_RUNG wire#w3
   RUNG wire#w1
      Contact( #DYNAMIC_DATA.msg_Flt_UnderRange )
      wire#w4
      Coil( #DYNAMIC_DATA.msg_Flt_OutOfRange )
   END_RUNG
   RUNG wire#w1
      Contact( #DYNAMIC_DATA.msg_Flt_OverRange )
   END_RUNG wire#w4
   // the same network as SCL:
   #_w1 := NOT #DYNAMIC_DATA.mode_SimOn OR #DYNAMIC_DATA.status_ConfigError;
   #DYNAMIC_DATA.msg_Flt_UnderRange := #_w1 AND ((#DYNAMIC_DATA.actual_Value < #DYNAMIC_DATA.cal_UR_Abs) OR #DYNAMIC_DATA.status_ConfigError);
   #DYNAMIC_DATA.msg_Flt_OverRange := #_w1 AND ((#DYNAMIC_DATA.actual_Value > #DYNAMIC_DATA.cal_OR_Abs) OR #DYNAMIC_DATA.status_ConfigError);
   #DYNAMIC_DATA.msg_Flt_OutOfRange := #_w1 AND (#DYNAMIC_DATA.msg_Flt_UnderRange OR #DYNAMIC_DATA.msg_Flt_OverRange);
END_REGION

REGION Network 22: IO evaluation — External fault detection
   // ▀▀▀▀▀▀▀▀▀▀▀▀▀▀▀▀▀▀▀▀▀▀▀▀▀▀▀▀▀▀▀▀▀▀▀▀▀▀▀▀▀▀▀▀
   // If the EXT_FAULT signal is active (EXT_FAULT = 1), activate the associated message signal
   // 
   // Note:    The signal is ignored if simulation mode is on
   // ▄▄▄▄▄▄▄▄▄▄▄▄▄▄▄▄▄▄▄▄▄▄▄▄▄▄▄▄▄▄▄▄▄▄▄▄▄▄▄▄▄▄▄▄
   RUNG wire#powerrail
      Contact( #EXT_FAULT )
      I_Contact( #DYNAMIC_DATA.mode_SimOn )
      Coil( #DYNAMIC_DATA.msg_Flt_External )
   END_RUNG
   // the same network as SCL:
   #DYNAMIC_DATA.msg_Flt_External := #EXT_FAULT AND NOT #DYNAMIC_DATA.mode_SimOn;
END_REGION

REGION Network 23: Operating mode — Simulation mode
   // ▀▀▀▀▀▀▀▀▀▀▀▀▀▀▀▀▀▀▀▀▀▀▀▀▀▀▀▀▀▀▀▀▀▀▀▀▀▀▀▀▀▀▀▀
   // If simulation mode is enabled (mode_SimOn = 1) and a configuration error is not present,
   // (status_ConfigError = 0) overwrite the actual_Value with the mode_SimValue signal set by the 
   // operator.
   // 
   // Note:    Any fault signals will be suppressed (turned off) is simulation mode is active
   //      and a configuration error is not present
   // 
   //      The simulated value (mode_SimValue) is restricted to the range given in 
   //      actual_AiScaleData.SCALE_MIN and actual_AiScaleData.SCALE_MAX
   // ▄▄▄▄▄▄▄▄▄▄▄▄▄▄▄▄▄▄▄▄▄▄▄▄▄▄▄▄▄▄▄▄▄▄▄▄▄▄▄▄▄▄▄▄
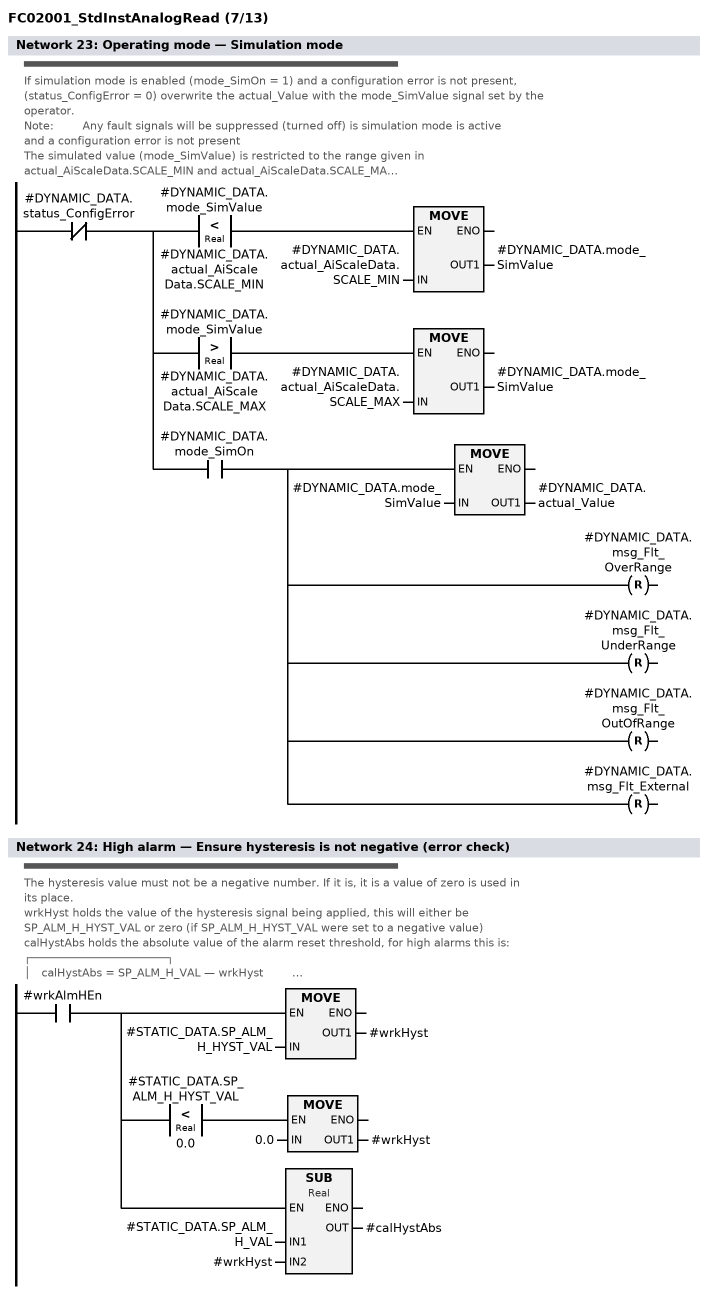
   RUNG wire#powerrail
      I_Contact( #DYNAMIC_DATA.status_ConfigError )
      wire#w1
      { S7_Templates := "SrcType := Real" } LT_Contact(in1 := #DYNAMIC_DATA.mode_SimValue, in2 := #DYNAMIC_DATA.actual_AiScaleData.SCALE_MIN)
      { S7_GenerateENO := "TRUE" } Move(in := #DYNAMIC_DATA.actual_AiScaleData.SCALE_MIN, out1 => #DYNAMIC_DATA.mode_SimValue)
   END_RUNG
   RUNG wire#w1
      { S7_Templates := "SrcType := Real" } GT_Contact(in1 := #DYNAMIC_DATA.mode_SimValue, in2 := #DYNAMIC_DATA.actual_AiScaleData.SCALE_MAX)
      { S7_GenerateENO := "TRUE" } Move(in := #DYNAMIC_DATA.actual_AiScaleData.SCALE_MAX, out1 => #DYNAMIC_DATA.mode_SimValue)
   END_RUNG
   RUNG wire#w1
      Contact( #DYNAMIC_DATA.mode_SimOn )
      wire#w2
      { S7_GenerateENO := "TRUE" } Move(in := #DYNAMIC_DATA.mode_SimValue, out1 => #DYNAMIC_DATA.actual_Value)
   END_RUNG
   RUNG wire#w2
      R_Coil( #DYNAMIC_DATA.msg_Flt_OverRange )
   END_RUNG
   RUNG wire#w2
      R_Coil( #DYNAMIC_DATA.msg_Flt_UnderRange )
   END_RUNG
   RUNG wire#w2
      R_Coil( #DYNAMIC_DATA.msg_Flt_OutOfRange )
   END_RUNG
   RUNG wire#w2
      R_Coil( #DYNAMIC_DATA.msg_Flt_External )
   END_RUNG
   // the same network as SCL:
   #_w1 := NOT #DYNAMIC_DATA.status_ConfigError;
   IF #_w1 AND (#DYNAMIC_DATA.mode_SimValue < #DYNAMIC_DATA.actual_AiScaleData.SCALE_MIN) THEN
       #DYNAMIC_DATA.mode_SimValue := #DYNAMIC_DATA.actual_AiScaleData.SCALE_MIN;
   END_IF;
   IF #_w1 AND (#DYNAMIC_DATA.mode_SimValue > #DYNAMIC_DATA.actual_AiScaleData.SCALE_MAX) THEN
       #DYNAMIC_DATA.mode_SimValue := #DYNAMIC_DATA.actual_AiScaleData.SCALE_MAX;
   END_IF;
   IF #_w1 AND #DYNAMIC_DATA.mode_SimOn THEN
       #DYNAMIC_DATA.actual_Value := #DYNAMIC_DATA.mode_SimValue;
       #DYNAMIC_DATA.msg_Flt_OverRange := FALSE;
       #DYNAMIC_DATA.msg_Flt_UnderRange := FALSE;
       #DYNAMIC_DATA.msg_Flt_OutOfRange := FALSE;
       #DYNAMIC_DATA.msg_Flt_External := FALSE;
   END_IF;
END_REGION

REGION Network 24: High alarm — Ensure hysteresis is not negative (error check)
   // ▀▀▀▀▀▀▀▀▀▀▀▀▀▀▀▀▀▀▀▀▀▀▀▀▀▀▀▀▀▀▀▀▀▀▀▀▀▀▀▀▀▀▀▀
   // The hysteresis value must not be a negative number. If it is, it is a value of zero is used in
   // its place.
   // 
   // wrkHyst holds the value of the hysteresis signal being applied, this will either be 
   // SP_ALM_H_HYST_VAL or zero (if SP_ALM_H_HYST_VAL were set to a negative value)
   // 
   // calHystAbs holds the absolute value of the alarm reset threshold, for high alarms this is:
   // ┌─────────────────────┐
   // │ calHystAbs = SP_ALM_H_VAL — wrkHyst      │
   // └─────────────────────┘
   // 
   // The two threshold values for the high alarm are thus:
   // 
   //      High alarm activation threshold = SP_ALM_H_VAL
   //      High alarm reset threshold          = calHystAbs
   // 
   // Note:    The hysteresis is only checked if alarm is being evaluated
   // ▄▄▄▄▄▄▄▄▄▄▄▄▄▄▄▄▄▄▄▄▄▄▄▄▄▄▄▄▄▄▄▄▄▄▄▄▄▄▄▄▄▄▄▄
   RUNG wire#powerrail
      Contact( #wrkAlmHEn )
      wire#w1
      { S7_GenerateENO := "TRUE" } Move(in := #STATIC_DATA.SP_ALM_H_HYST_VAL, out1 => #wrkHyst)
   END_RUNG
   RUNG wire#w1
      { S7_Templates := "SrcType := Real" } LT_Contact(in1 := #STATIC_DATA.SP_ALM_H_HYST_VAL, in2 := 0.0)
      { S7_GenerateENO := "TRUE" } Move(in := 0.0, out1 => #wrkHyst)
   END_RUNG
   RUNG wire#w1
      { S7_Templates := "SrcType := Real"; S7_GenerateENO := "TRUE" } Sub(in1 := #STATIC_DATA.SP_ALM_H_VAL, in2 := #wrkHyst, out => #calHystAbs)
   END_RUNG
   // the same network as SCL:
   IF #wrkAlmHEn THEN #wrkHyst := #STATIC_DATA.SP_ALM_H_HYST_VAL; END_IF;
   IF #wrkAlmHEn AND (#STATIC_DATA.SP_ALM_H_HYST_VAL < 0.0) THEN #wrkHyst := 0.0; END_IF;
   IF #wrkAlmHEn THEN #calHystAbs := #STATIC_DATA.SP_ALM_H_VAL - #wrkHyst; END_IF;
END_REGION

REGION Network 25: High alarm — Check for activation level and ON-DELAY timer
   // ▀▀▀▀▀▀▀▀▀▀▀▀▀▀▀▀▀▀▀▀▀▀▀▀▀▀▀▀▀▀▀▀▀▀▀▀▀▀▀▀▀▀▀▀
   // If the high alarm has been enabled and is not masked and the actual_Value is greater than or 
   // equal to the alarm setpoint (SP_ALM_H_VAL), but the alarm has not yet been triggered 
   // (msg_Alm_H = 0) then the ON-DELAY phase is active (the alarm timer is counting down).
   // 
   // The timer will begin to count down from the value in TIME_ALM_H_ON_DEL using the 200ms 
   // pulse (it will count down in increments of 0.2s). If the high alarm timer is less than or equal to 
   // zero, then the ON-DELAY has expired and the High Alarm message will become active.
   // 
   // If at any point during the ON-DELAY count down, the actual_Value drops below the activation
   // setpoint (SP_ALM_H_VAL), the timer will be reset to the TIME_ALM_H_ON_DEL value, forcing 
   // the ON-DELAY to start again.
   // ▄▄▄▄▄▄▄▄▄▄▄▄▄▄▄▄▄▄▄▄▄▄▄▄▄▄▄▄▄▄▄▄▄▄▄▄▄▄▄▄▄▄▄▄
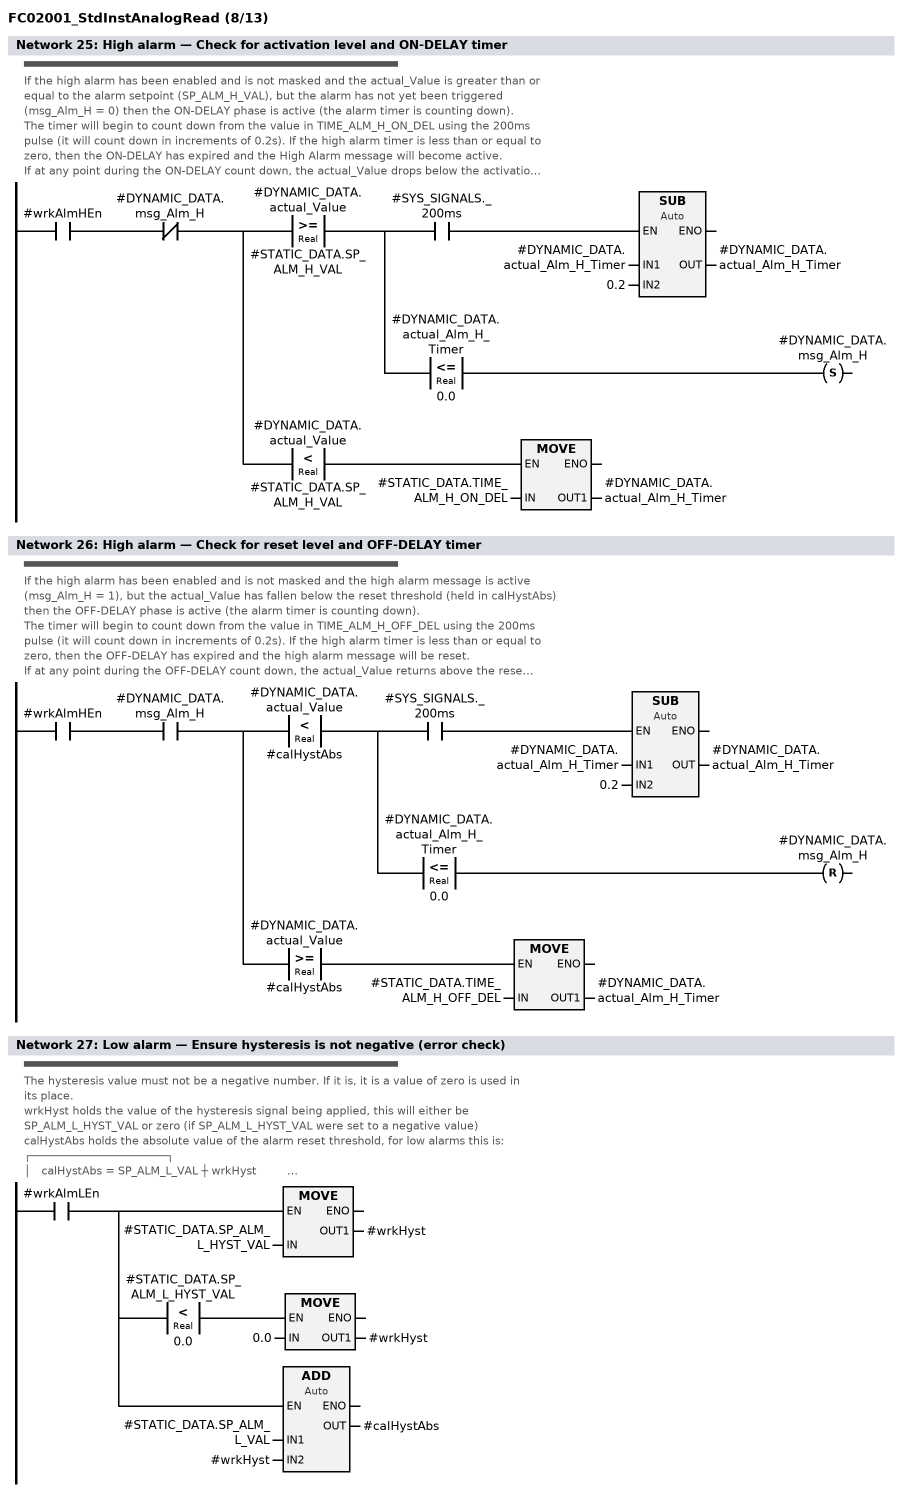
   RUNG wire#powerrail
      Contact( #wrkAlmHEn )
      I_Contact( #DYNAMIC_DATA.msg_Alm_H )
      wire#w1
      { S7_Templates := "SrcType := Real" } GE_Contact(in1 := #DYNAMIC_DATA.actual_Value, in2 := #STATIC_DATA.SP_ALM_H_VAL)
      wire#w2
      Contact( #SYS_SIGNALS._200ms )
      Sub(in1 := #DYNAMIC_DATA.actual_Alm_H_Timer, in2 := 0.2, out => #DYNAMIC_DATA.actual_Alm_H_Timer)
   END_RUNG
   RUNG wire#w2
      { S7_Templates := "SrcType := Real" } LE_Contact(in1 := #DYNAMIC_DATA.actual_Alm_H_Timer, in2 := 0.0)
      S_Coil( #DYNAMIC_DATA.msg_Alm_H )
   END_RUNG
   RUNG wire#w1
      { S7_Templates := "SrcType := Real" } LT_Contact(in1 := #DYNAMIC_DATA.actual_Value, in2 := #STATIC_DATA.SP_ALM_H_VAL)
      { S7_GenerateENO := "TRUE" } Move(in := #STATIC_DATA.TIME_ALM_H_ON_DEL, out1 => #DYNAMIC_DATA.actual_Alm_H_Timer)
   END_RUNG
   // the same network as SCL:
   #_w1 := #wrkAlmHEn AND NOT #DYNAMIC_DATA.msg_Alm_H;
   #_w2 := #_w1 AND (#DYNAMIC_DATA.actual_Value >= #STATIC_DATA.SP_ALM_H_VAL);
   IF #_w2 AND #SYS_SIGNALS._200ms THEN
       #DYNAMIC_DATA.actual_Alm_H_Timer := #DYNAMIC_DATA.actual_Alm_H_Timer - 0.2;
   END_IF;
   IF #_w2 AND (#DYNAMIC_DATA.actual_Alm_H_Timer <= 0.0) THEN #DYNAMIC_DATA.msg_Alm_H := TRUE; END_IF;
   IF #_w1 AND (#DYNAMIC_DATA.actual_Value < #STATIC_DATA.SP_ALM_H_VAL) THEN
       #DYNAMIC_DATA.actual_Alm_H_Timer := #STATIC_DATA.TIME_ALM_H_ON_DEL;
   END_IF;
END_REGION

REGION Network 26: High alarm — Check for reset level and OFF-DELAY timer
   // ▀▀▀▀▀▀▀▀▀▀▀▀▀▀▀▀▀▀▀▀▀▀▀▀▀▀▀▀▀▀▀▀▀▀▀▀▀▀▀▀▀▀▀▀
   // If the high alarm has been enabled and is not masked and the high alarm message is active 
   // (msg_Alm_H = 1), but the actual_Value has fallen below the reset threshold (held in calHystAbs) 
   // then the OFF-DELAY phase is active (the alarm timer is counting down).
   // 
   // The timer will begin to count down from the value in TIME_ALM_H_OFF_DEL using the 200ms 
   // pulse (it will count down in increments of 0.2s). If the high alarm timer is less than or equal to 
   // zero, then the OFF-DELAY has expired and the high alarm message will be reset.
   // 
   // If at any point during the OFF-DELAY count down, the actual_Value returns above the reset
   // threshold (calHystAbs), the timer will be reset to the TIME_ALM_H_OFF_DEL value, forcing 
   // the OFF-DELAY to start again.
   // ▄▄▄▄▄▄▄▄▄▄▄▄▄▄▄▄▄▄▄▄▄▄▄▄▄▄▄▄▄▄▄▄▄▄▄▄▄▄▄▄▄▄▄▄
   RUNG wire#powerrail
      Contact( #wrkAlmHEn )
      Contact( #DYNAMIC_DATA.msg_Alm_H )
      wire#w1
      { S7_Templates := "SrcType := Real" } LT_Contact(in1 := #DYNAMIC_DATA.actual_Value, in2 := #calHystAbs)
      wire#w2
      Contact( #SYS_SIGNALS._200ms )
      Sub(in1 := #DYNAMIC_DATA.actual_Alm_H_Timer, in2 := 0.2, out => #DYNAMIC_DATA.actual_Alm_H_Timer)
   END_RUNG
   RUNG wire#w2
      { S7_Templates := "SrcType := Real" } LE_Contact(in1 := #DYNAMIC_DATA.actual_Alm_H_Timer, in2 := 0.0)
      R_Coil( #DYNAMIC_DATA.msg_Alm_H )
   END_RUNG
   RUNG wire#w1
      { S7_Templates := "SrcType := Real" } GE_Contact(in1 := #DYNAMIC_DATA.actual_Value, in2 := #calHystAbs)
      { S7_GenerateENO := "TRUE" } Move(in := #STATIC_DATA.TIME_ALM_H_OFF_DEL, out1 => #DYNAMIC_DATA.actual_Alm_H_Timer)
   END_RUNG
   // the same network as SCL:
   #_w1 := #wrkAlmHEn AND #DYNAMIC_DATA.msg_Alm_H;
   #_w2 := #_w1 AND (#DYNAMIC_DATA.actual_Value < #calHystAbs);
   IF #_w2 AND #SYS_SIGNALS._200ms THEN
       #DYNAMIC_DATA.actual_Alm_H_Timer := #DYNAMIC_DATA.actual_Alm_H_Timer - 0.2;
   END_IF;
   IF #_w2 AND (#DYNAMIC_DATA.actual_Alm_H_Timer <= 0.0) THEN #DYNAMIC_DATA.msg_Alm_H := FALSE; END_IF;
   IF #_w1 AND (#DYNAMIC_DATA.actual_Value >= #calHystAbs) THEN
       #DYNAMIC_DATA.actual_Alm_H_Timer := #STATIC_DATA.TIME_ALM_H_OFF_DEL;
   END_IF;
END_REGION

REGION Network 27: Low alarm — Ensure hysteresis is not negative (error check)
   // ▀▀▀▀▀▀▀▀▀▀▀▀▀▀▀▀▀▀▀▀▀▀▀▀▀▀▀▀▀▀▀▀▀▀▀▀▀▀▀▀▀▀▀▀
   // The hysteresis value must not be a negative number. If it is, it is a value of zero is used in
   // its place.
   // 
   // wrkHyst holds the value of the hysteresis signal being applied, this will either be 
   // SP_ALM_L_HYST_VAL or zero (if SP_ALM_L_HYST_VAL were set to a negative value)
   // 
   // calHystAbs holds the absolute value of the alarm reset threshold, for low alarms this is:
   // ┌─────────────────────┐
   // │ calHystAbs = SP_ALM_L_VAL ┼ wrkHyst       │
   // └─────────────────────┘
   // 
   // The two threshold values for the low alarm are thus:
   // 
   //      Low alarm activation threshold = SP_ALM_L_VAL
   //      Low alarm reset threshold          = calHystAbs
   // 
   // Note:    The hysteresis is only checked if alarm is being evaluated
   // ▄▄▄▄▄▄▄▄▄▄▄▄▄▄▄▄▄▄▄▄▄▄▄▄▄▄▄▄▄▄▄▄▄▄▄▄▄▄▄▄▄▄▄▄
   RUNG wire#powerrail
      Contact( #wrkAlmLEn )
      wire#w1
      { S7_GenerateENO := "TRUE" } Move(in := #STATIC_DATA.SP_ALM_L_HYST_VAL, out1 => #wrkHyst)
   END_RUNG
   RUNG wire#w1
      { S7_Templates := "SrcType := Real" } LT_Contact(in1 := #STATIC_DATA.SP_ALM_L_HYST_VAL, in2 := 0.0)
      { S7_GenerateENO := "TRUE" } Move(in := 0.0, out1 => #wrkHyst)
   END_RUNG
   RUNG wire#w1
      Add(in1 := #STATIC_DATA.SP_ALM_L_VAL, in2 := #wrkHyst, out => #calHystAbs)
   END_RUNG
   // the same network as SCL:
   IF #wrkAlmLEn THEN #wrkHyst := #STATIC_DATA.SP_ALM_L_HYST_VAL; END_IF;
   IF #wrkAlmLEn AND (#STATIC_DATA.SP_ALM_L_HYST_VAL < 0.0) THEN #wrkHyst := 0.0; END_IF;
   IF #wrkAlmLEn THEN #calHystAbs := #STATIC_DATA.SP_ALM_L_VAL + #wrkHyst; END_IF;
END_REGION

REGION Network 28: Low alarm — Check for activation level and ON-DELAY timer
   // ▀▀▀▀▀▀▀▀▀▀▀▀▀▀▀▀▀▀▀▀▀▀▀▀▀▀▀▀▀▀▀▀▀▀▀▀▀▀▀▀▀▀▀▀
   // If the low alarm has been enabled and is not masked and the actual_Value is less than or 
   // equal to the alarm setpoint (SP_ALM_L_VAL), but the alarm has not yet been triggered 
   // (msg_Alm_L = 0) then the ON-DELAY phase is active (the alarm timer is counting down).
   // 
   // The timer will begin to count down from the value in TIME_ALM_L_ON_DEL using the 200ms 
   // pulse (it will count down in increments of 0.2s). If the Low alarm timer is less than or equal to 
   // zero, then the ON-DELAY has expired and the Low Alarm message will become active.
   // 
   // If at any point during the ON-DELAY count down, the actual_Value rises above the activation
   // setpoint (SP_ALM_L_VAL), the timer will be reset to the TIME_ALM_L_ON_DEL value, forcing 
   // the ON-DELAY to start again.
   // ▄▄▄▄▄▄▄▄▄▄▄▄▄▄▄▄▄▄▄▄▄▄▄▄▄▄▄▄▄▄▄▄▄▄▄▄▄▄▄▄▄▄▄▄
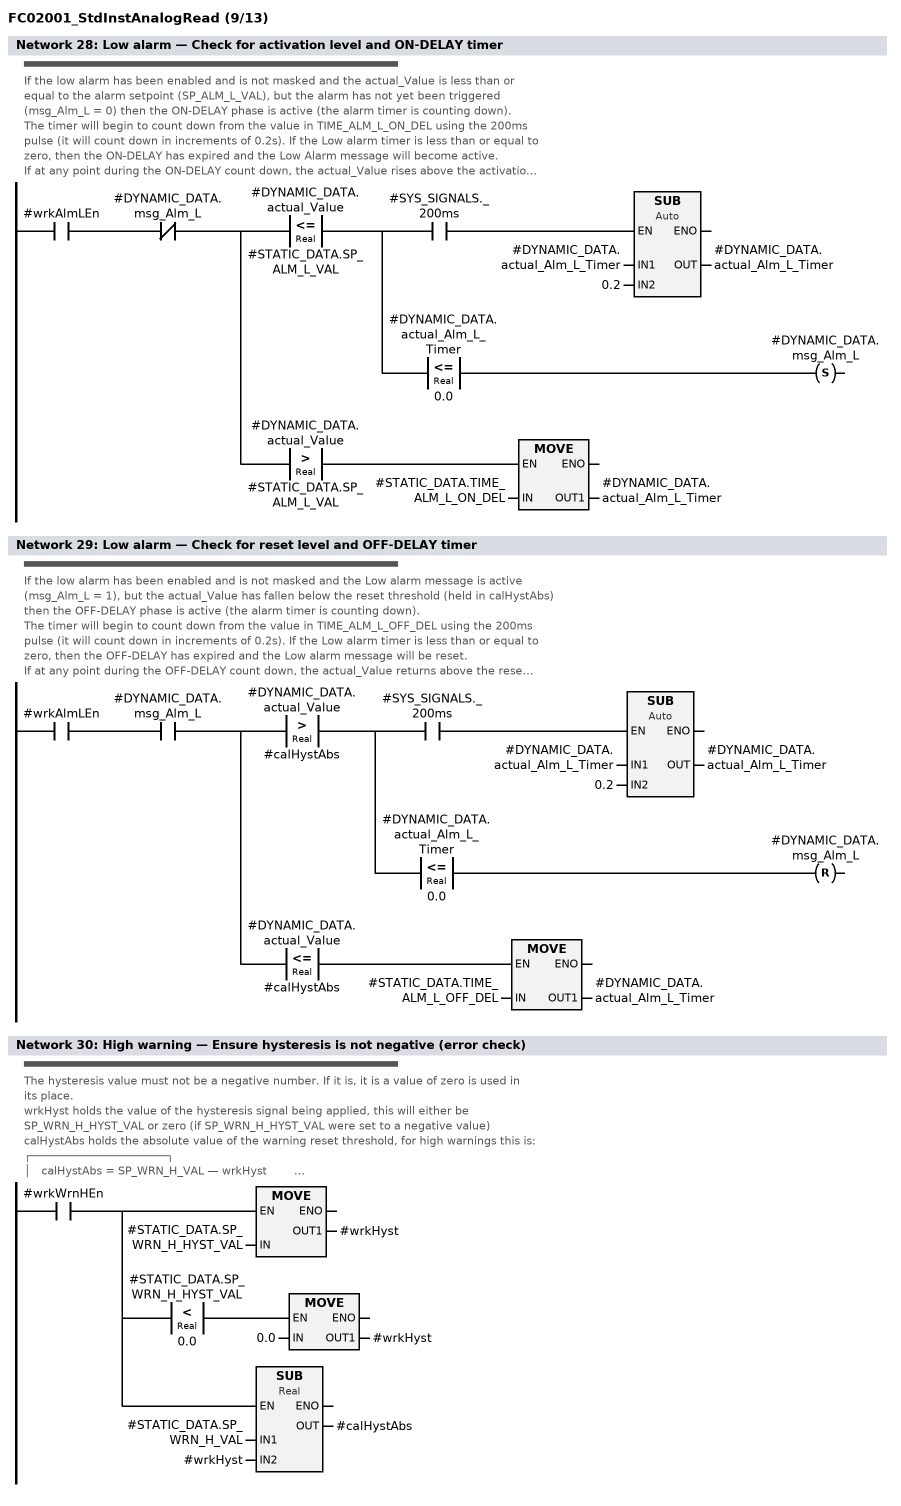
   RUNG wire#powerrail
      Contact( #wrkAlmLEn )
      I_Contact( #DYNAMIC_DATA.msg_Alm_L )
      wire#w1
      { S7_Templates := "SrcType := Real" } LE_Contact(in1 := #DYNAMIC_DATA.actual_Value, in2 := #STATIC_DATA.SP_ALM_L_VAL)
      wire#w2
      Contact( #SYS_SIGNALS._200ms )
      Sub(in1 := #DYNAMIC_DATA.actual_Alm_L_Timer, in2 := 0.2, out => #DYNAMIC_DATA.actual_Alm_L_Timer)
   END_RUNG
   RUNG wire#w2
      { S7_Templates := "SrcType := Real" } LE_Contact(in1 := #DYNAMIC_DATA.actual_Alm_L_Timer, in2 := 0.0)
      S_Coil( #DYNAMIC_DATA.msg_Alm_L )
   END_RUNG
   RUNG wire#w1
      { S7_Templates := "SrcType := Real" } GT_Contact(in1 := #DYNAMIC_DATA.actual_Value, in2 := #STATIC_DATA.SP_ALM_L_VAL)
      { S7_GenerateENO := "TRUE" } Move(in := #STATIC_DATA.TIME_ALM_L_ON_DEL, out1 => #DYNAMIC_DATA.actual_Alm_L_Timer)
   END_RUNG
   // the same network as SCL:
   #_w1 := #wrkAlmLEn AND NOT #DYNAMIC_DATA.msg_Alm_L;
   #_w2 := #_w1 AND (#DYNAMIC_DATA.actual_Value <= #STATIC_DATA.SP_ALM_L_VAL);
   IF #_w2 AND #SYS_SIGNALS._200ms THEN
       #DYNAMIC_DATA.actual_Alm_L_Timer := #DYNAMIC_DATA.actual_Alm_L_Timer - 0.2;
   END_IF;
   IF #_w2 AND (#DYNAMIC_DATA.actual_Alm_L_Timer <= 0.0) THEN #DYNAMIC_DATA.msg_Alm_L := TRUE; END_IF;
   IF #_w1 AND (#DYNAMIC_DATA.actual_Value > #STATIC_DATA.SP_ALM_L_VAL) THEN
       #DYNAMIC_DATA.actual_Alm_L_Timer := #STATIC_DATA.TIME_ALM_L_ON_DEL;
   END_IF;
END_REGION

REGION Network 29: Low alarm — Check for reset level and OFF-DELAY timer
   // ▀▀▀▀▀▀▀▀▀▀▀▀▀▀▀▀▀▀▀▀▀▀▀▀▀▀▀▀▀▀▀▀▀▀▀▀▀▀▀▀▀▀▀▀
   // If the low alarm has been enabled and is not masked and the Low alarm message is active 
   // (msg_Alm_L = 1), but the actual_Value has fallen below the reset threshold (held in calHystAbs) 
   // then the OFF-DELAY phase is active (the alarm timer is counting down).
   // 
   // The timer will begin to count down from the value in TIME_ALM_L_OFF_DEL using the 200ms 
   // pulse (it will count down in increments of 0.2s). If the Low alarm timer is less than or equal to 
   // zero, then the OFF-DELAY has expired and the Low alarm message will be reset.
   // 
   // If at any point during the OFF-DELAY count down, the actual_Value returns above the reset
   // threshold (calHystAbs), the timer will be reset to the TIME_ALM_L_OFF_DEL value, forcing 
   // the OFF-DELAY to start again.
   // ▄▄▄▄▄▄▄▄▄▄▄▄▄▄▄▄▄▄▄▄▄▄▄▄▄▄▄▄▄▄▄▄▄▄▄▄▄▄▄▄▄▄▄▄
   RUNG wire#powerrail
      Contact( #wrkAlmLEn )
      Contact( #DYNAMIC_DATA.msg_Alm_L )
      wire#w1
      { S7_Templates := "SrcType := Real" } GT_Contact(in1 := #DYNAMIC_DATA.actual_Value, in2 := #calHystAbs)
      wire#w2
      Contact( #SYS_SIGNALS._200ms )
      Sub(in1 := #DYNAMIC_DATA.actual_Alm_L_Timer, in2 := 0.2, out => #DYNAMIC_DATA.actual_Alm_L_Timer)
   END_RUNG
   RUNG wire#w2
      { S7_Templates := "SrcType := Real" } LE_Contact(in1 := #DYNAMIC_DATA.actual_Alm_L_Timer, in2 := 0.0)
      R_Coil( #DYNAMIC_DATA.msg_Alm_L )
   END_RUNG
   RUNG wire#w1
      { S7_Templates := "SrcType := Real" } LE_Contact(in1 := #DYNAMIC_DATA.actual_Value, in2 := #calHystAbs)
      { S7_GenerateENO := "TRUE" } Move(in := #STATIC_DATA.TIME_ALM_L_OFF_DEL, out1 => #DYNAMIC_DATA.actual_Alm_L_Timer)
   END_RUNG
   // the same network as SCL:
   #_w1 := #wrkAlmLEn AND #DYNAMIC_DATA.msg_Alm_L;
   #_w2 := #_w1 AND (#DYNAMIC_DATA.actual_Value > #calHystAbs);
   IF #_w2 AND #SYS_SIGNALS._200ms THEN
       #DYNAMIC_DATA.actual_Alm_L_Timer := #DYNAMIC_DATA.actual_Alm_L_Timer - 0.2;
   END_IF;
   IF #_w2 AND (#DYNAMIC_DATA.actual_Alm_L_Timer <= 0.0) THEN #DYNAMIC_DATA.msg_Alm_L := FALSE; END_IF;
   IF #_w1 AND (#DYNAMIC_DATA.actual_Value <= #calHystAbs) THEN
       #DYNAMIC_DATA.actual_Alm_L_Timer := #STATIC_DATA.TIME_ALM_L_OFF_DEL;
   END_IF;
END_REGION

REGION Network 30: High warning — Ensure hysteresis is not negative (error check)
   // ▀▀▀▀▀▀▀▀▀▀▀▀▀▀▀▀▀▀▀▀▀▀▀▀▀▀▀▀▀▀▀▀▀▀▀▀▀▀▀▀▀▀▀▀
   // The hysteresis value must not be a negative number. If it is, it is a value of zero is used in
   // its place.
   // 
   // wrkHyst holds the value of the hysteresis signal being applied, this will either be 
   // SP_WRN_H_HYST_VAL or zero (if SP_WRN_H_HYST_VAL were set to a negative value)
   // 
   // calHystAbs holds the absolute value of the warning reset threshold, for high warnings this is:
   // ┌─────────────────────┐
   // │ calHystAbs = SP_WRN_H_VAL — wrkHyst      │
   // └─────────────────────┘
   // 
   // The two threshold values for the high warning are thus:
   // 
   //      High warning activation threshold = SP_WRN_H_VAL
   //      High warning reset threshold          = calHystAbs
   // 
   // Note:    The hysteresis is only checked if warning is being evaluated
   // ▄▄▄▄▄▄▄▄▄▄▄▄▄▄▄▄▄▄▄▄▄▄▄▄▄▄▄▄▄▄▄▄▄▄▄▄▄▄▄▄▄▄▄▄
   RUNG wire#powerrail
      Contact( #wrkWrnHEn )
      wire#w1
      { S7_GenerateENO := "TRUE" } Move(in := #STATIC_DATA.SP_WRN_H_HYST_VAL, out1 => #wrkHyst)
   END_RUNG
   RUNG wire#w1
      { S7_Templates := "SrcType := Real" } LT_Contact(in1 := #STATIC_DATA.SP_WRN_H_HYST_VAL, in2 := 0.0)
      { S7_GenerateENO := "TRUE" } Move(in := 0.0, out1 => #wrkHyst)
   END_RUNG
   RUNG wire#w1
      { S7_Templates := "SrcType := Real"; S7_GenerateENO := "TRUE" } Sub(in1 := #STATIC_DATA.SP_WRN_H_VAL, in2 := #wrkHyst, out => #calHystAbs)
   END_RUNG
   // the same network as SCL:
   IF #wrkWrnHEn THEN #wrkHyst := #STATIC_DATA.SP_WRN_H_HYST_VAL; END_IF;
   IF #wrkWrnHEn AND (#STATIC_DATA.SP_WRN_H_HYST_VAL < 0.0) THEN #wrkHyst := 0.0; END_IF;
   IF #wrkWrnHEn THEN #calHystAbs := #STATIC_DATA.SP_WRN_H_VAL - #wrkHyst; END_IF;
END_REGION

REGION Network 31: High warning — Check for activation level and ON-DELAY timer
   // ▀▀▀▀▀▀▀▀▀▀▀▀▀▀▀▀▀▀▀▀▀▀▀▀▀▀▀▀▀▀▀▀▀▀▀▀▀▀▀▀▀▀▀▀
   // If the high warning has been enabled and is not masked and the actual_Value is greater than or 
   // equal to the warning setpoint (SP_WRN_H_VAL), but the warning has not yet been triggered 
   // (msg_Wrn_H = 0) then the ON-DELAY phase is active (the warning timer is counting down).
   // 
   // The timer will begin to count down from the value in TIME_WRN_H_ON_DEL using the 200ms 
   // pulse (it will count down in increments of 0.2s). If the high warning timer is less than or equal to 
   // zero, then the ON-DELAY has expired and the High warning message will become active.
   // 
   // If at any point during the ON-DELAY count down, the actual_Value drops below the activation
   // setpoint (SP_WRN_H_VAL), the timer will be reset to the TIME_WRN_H_ON_DEL value, forcing 
   // the ON-DELAY to start again.
   // ▄▄▄▄▄▄▄▄▄▄▄▄▄▄▄▄▄▄▄▄▄▄▄▄▄▄▄▄▄▄▄▄▄▄▄▄▄▄▄▄▄▄▄▄
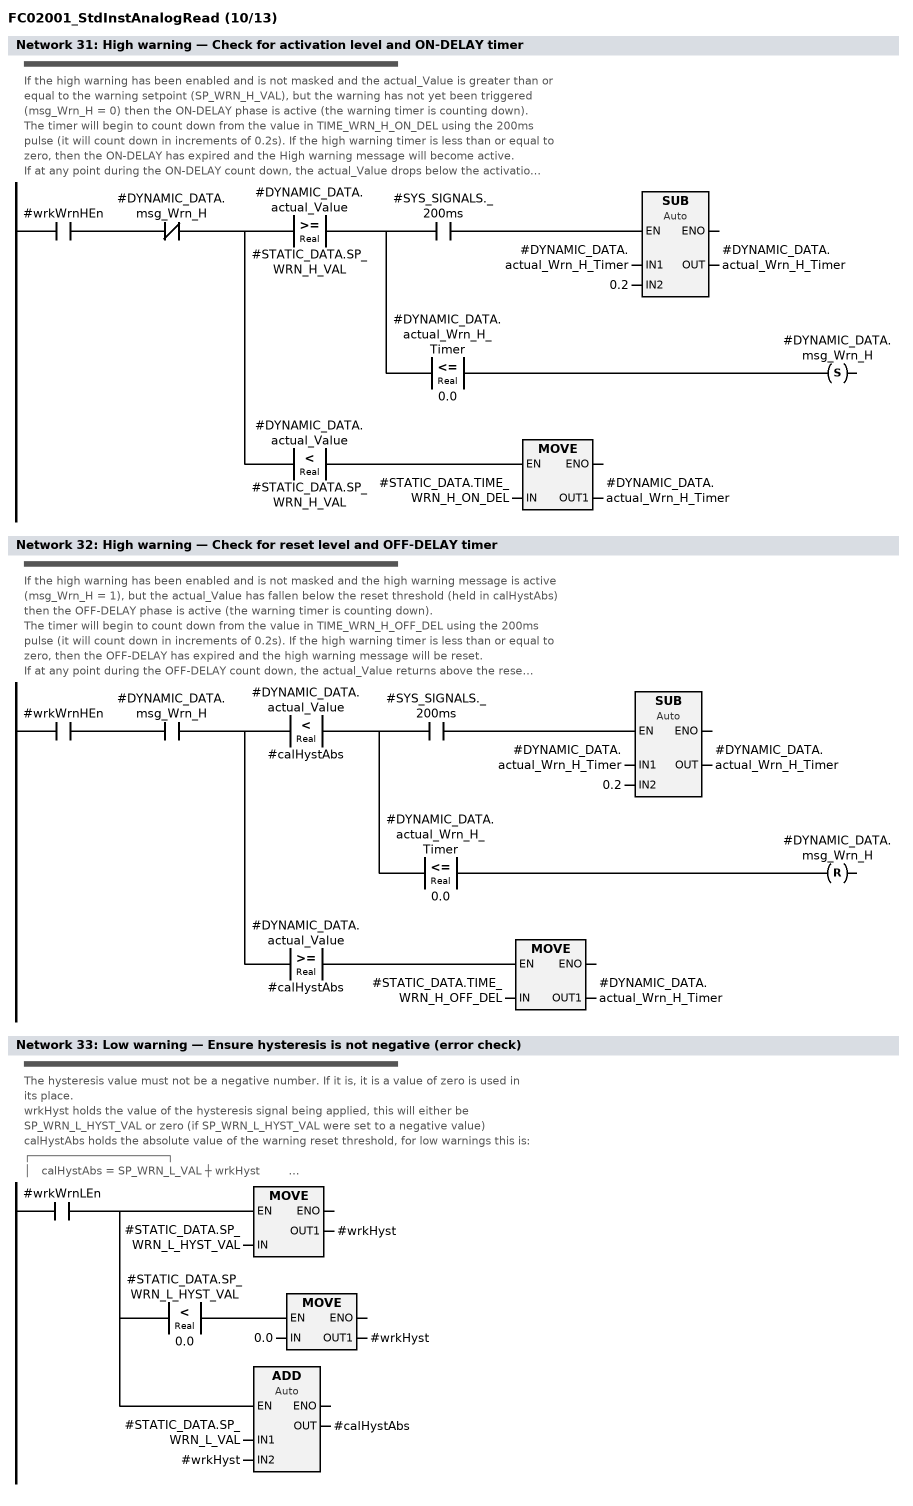
   RUNG wire#powerrail
      Contact( #wrkWrnHEn )
      I_Contact( #DYNAMIC_DATA.msg_Wrn_H )
      wire#w1
      { S7_Templates := "SrcType := Real" } GE_Contact(in1 := #DYNAMIC_DATA.actual_Value, in2 := #STATIC_DATA.SP_WRN_H_VAL)
      wire#w2
      Contact( #SYS_SIGNALS._200ms )
      Sub(in1 := #DYNAMIC_DATA.actual_Wrn_H_Timer, in2 := 0.2, out => #DYNAMIC_DATA.actual_Wrn_H_Timer)
   END_RUNG
   RUNG wire#w2
      { S7_Templates := "SrcType := Real" } LE_Contact(in1 := #DYNAMIC_DATA.actual_Wrn_H_Timer, in2 := 0.0)
      S_Coil( #DYNAMIC_DATA.msg_Wrn_H )
   END_RUNG
   RUNG wire#w1
      { S7_Templates := "SrcType := Real" } LT_Contact(in1 := #DYNAMIC_DATA.actual_Value, in2 := #STATIC_DATA.SP_WRN_H_VAL)
      { S7_GenerateENO := "TRUE" } Move(in := #STATIC_DATA.TIME_WRN_H_ON_DEL, out1 => #DYNAMIC_DATA.actual_Wrn_H_Timer)
   END_RUNG
   // the same network as SCL:
   #_w1 := #wrkWrnHEn AND NOT #DYNAMIC_DATA.msg_Wrn_H;
   #_w2 := #_w1 AND (#DYNAMIC_DATA.actual_Value >= #STATIC_DATA.SP_WRN_H_VAL);
   IF #_w2 AND #SYS_SIGNALS._200ms THEN
       #DYNAMIC_DATA.actual_Wrn_H_Timer := #DYNAMIC_DATA.actual_Wrn_H_Timer - 0.2;
   END_IF;
   IF #_w2 AND (#DYNAMIC_DATA.actual_Wrn_H_Timer <= 0.0) THEN #DYNAMIC_DATA.msg_Wrn_H := TRUE; END_IF;
   IF #_w1 AND (#DYNAMIC_DATA.actual_Value < #STATIC_DATA.SP_WRN_H_VAL) THEN
       #DYNAMIC_DATA.actual_Wrn_H_Timer := #STATIC_DATA.TIME_WRN_H_ON_DEL;
   END_IF;
END_REGION

REGION Network 32: High warning — Check for reset level and OFF-DELAY timer
   // ▀▀▀▀▀▀▀▀▀▀▀▀▀▀▀▀▀▀▀▀▀▀▀▀▀▀▀▀▀▀▀▀▀▀▀▀▀▀▀▀▀▀▀▀
   // If the high warning has been enabled and is not masked and the high warning message is active 
   // (msg_Wrn_H = 1), but the actual_Value has fallen below the reset threshold (held in calHystAbs) 
   // then the OFF-DELAY phase is active (the warning timer is counting down).
   // 
   // The timer will begin to count down from the value in TIME_WRN_H_OFF_DEL using the 200ms 
   // pulse (it will count down in increments of 0.2s). If the high warning timer is less than or equal to 
   // zero, then the OFF-DELAY has expired and the high warning message will be reset.
   // 
   // If at any point during the OFF-DELAY count down, the actual_Value returns above the reset
   // threshold (calHystAbs), the timer will be reset to the TIME_WRN_H_OFF_DEL value, forcing 
   // the OFF-DELAY to start again.
   // ▄▄▄▄▄▄▄▄▄▄▄▄▄▄▄▄▄▄▄▄▄▄▄▄▄▄▄▄▄▄▄▄▄▄▄▄▄▄▄▄▄▄▄▄
   RUNG wire#powerrail
      Contact( #wrkWrnHEn )
      Contact( #DYNAMIC_DATA.msg_Wrn_H )
      wire#w1
      { S7_Templates := "SrcType := Real" } LT_Contact(in1 := #DYNAMIC_DATA.actual_Value, in2 := #calHystAbs)
      wire#w2
      Contact( #SYS_SIGNALS._200ms )
      Sub(in1 := #DYNAMIC_DATA.actual_Wrn_H_Timer, in2 := 0.2, out => #DYNAMIC_DATA.actual_Wrn_H_Timer)
   END_RUNG
   RUNG wire#w2
      { S7_Templates := "SrcType := Real" } LE_Contact(in1 := #DYNAMIC_DATA.actual_Wrn_H_Timer, in2 := 0.0)
      R_Coil( #DYNAMIC_DATA.msg_Wrn_H )
   END_RUNG
   RUNG wire#w1
      { S7_Templates := "SrcType := Real" } GE_Contact(in1 := #DYNAMIC_DATA.actual_Value, in2 := #calHystAbs)
      { S7_GenerateENO := "TRUE" } Move(in := #STATIC_DATA.TIME_WRN_H_OFF_DEL, out1 => #DYNAMIC_DATA.actual_Wrn_H_Timer)
   END_RUNG
   // the same network as SCL:
   #_w1 := #wrkWrnHEn AND #DYNAMIC_DATA.msg_Wrn_H;
   #_w2 := #_w1 AND (#DYNAMIC_DATA.actual_Value < #calHystAbs);
   IF #_w2 AND #SYS_SIGNALS._200ms THEN
       #DYNAMIC_DATA.actual_Wrn_H_Timer := #DYNAMIC_DATA.actual_Wrn_H_Timer - 0.2;
   END_IF;
   IF #_w2 AND (#DYNAMIC_DATA.actual_Wrn_H_Timer <= 0.0) THEN #DYNAMIC_DATA.msg_Wrn_H := FALSE; END_IF;
   IF #_w1 AND (#DYNAMIC_DATA.actual_Value >= #calHystAbs) THEN
       #DYNAMIC_DATA.actual_Wrn_H_Timer := #STATIC_DATA.TIME_WRN_H_OFF_DEL;
   END_IF;
END_REGION

REGION Network 33: Low warning — Ensure hysteresis is not negative (error check)
   // ▀▀▀▀▀▀▀▀▀▀▀▀▀▀▀▀▀▀▀▀▀▀▀▀▀▀▀▀▀▀▀▀▀▀▀▀▀▀▀▀▀▀▀▀
   // The hysteresis value must not be a negative number. If it is, it is a value of zero is used in
   // its place.
   // 
   // wrkHyst holds the value of the hysteresis signal being applied, this will either be 
   // SP_WRN_L_HYST_VAL or zero (if SP_WRN_L_HYST_VAL were set to a negative value)
   // 
   // calHystAbs holds the absolute value of the warning reset threshold, for low warnings this is:
   // ┌─────────────────────┐
   // │ calHystAbs = SP_WRN_L_VAL ┼ wrkHyst      │
   // └─────────────────────┘
   // 
   // The two threshold values for the low warning are thus:
   // 
   //      Low warning activation threshold = SP_WRN_L_VAL
   //      Low warning reset threshold          = calHystAbs
   // 
   // Note:    The hysteresis is only checked if warning is being evaluated
   // ▄▄▄▄▄▄▄▄▄▄▄▄▄▄▄▄▄▄▄▄▄▄▄▄▄▄▄▄▄▄▄▄▄▄▄▄▄▄▄▄▄▄▄▄
   RUNG wire#powerrail
      Contact( #wrkWrnLEn )
      wire#w1
      { S7_GenerateENO := "TRUE" } Move(in := #STATIC_DATA.SP_WRN_L_HYST_VAL, out1 => #wrkHyst)
   END_RUNG
   RUNG wire#w1
      { S7_Templates := "SrcType := Real" } LT_Contact(in1 := #STATIC_DATA.SP_WRN_L_HYST_VAL, in2 := 0.0)
      { S7_GenerateENO := "TRUE" } Move(in := 0.0, out1 => #wrkHyst)
   END_RUNG
   RUNG wire#w1
      Add(in1 := #STATIC_DATA.SP_WRN_L_VAL, in2 := #wrkHyst, out => #calHystAbs)
   END_RUNG
   // the same network as SCL:
   IF #wrkWrnLEn THEN #wrkHyst := #STATIC_DATA.SP_WRN_L_HYST_VAL; END_IF;
   IF #wrkWrnLEn AND (#STATIC_DATA.SP_WRN_L_HYST_VAL < 0.0) THEN #wrkHyst := 0.0; END_IF;
   IF #wrkWrnLEn THEN #calHystAbs := #STATIC_DATA.SP_WRN_L_VAL + #wrkHyst; END_IF;
END_REGION

REGION Network 34: Low warning — Check for activation level and ON-DELAY timer
   // ▀▀▀▀▀▀▀▀▀▀▀▀▀▀▀▀▀▀▀▀▀▀▀▀▀▀▀▀▀▀▀▀▀▀▀▀▀▀▀▀▀▀▀▀
   // If the low warning has been enabled and is not masked and the actual_Value is less than or 
   // equal to the warning setpoint (SP_WRN_L_VAL), but the warning has not yet been triggered 
   // (msg_Wrn_L = 0) then the ON-DELAY phase is active (the warning timer is counting down).
   // 
   // The timer will begin to count down from the value in TIME_WRN_L_ON_DEL using the 200ms 
   // pulse (it will count down in increments of 0.2s). If the Low warning timer is less than or equal to 
   // zero, then the ON-DELAY has expired and the Low Warning message will become active.
   // 
   // If at any point during the ON-DELAY count down, the actual_Value rises above the activation
   // setpoint (SP_WRN_L_VAL), the timer will be reset to the TIME_WRN_L_ON_DEL value, forcing 
   // the ON-DELAY to start again.
   // ▄▄▄▄▄▄▄▄▄▄▄▄▄▄▄▄▄▄▄▄▄▄▄▄▄▄▄▄▄▄▄▄▄▄▄▄▄▄▄▄▄▄▄▄
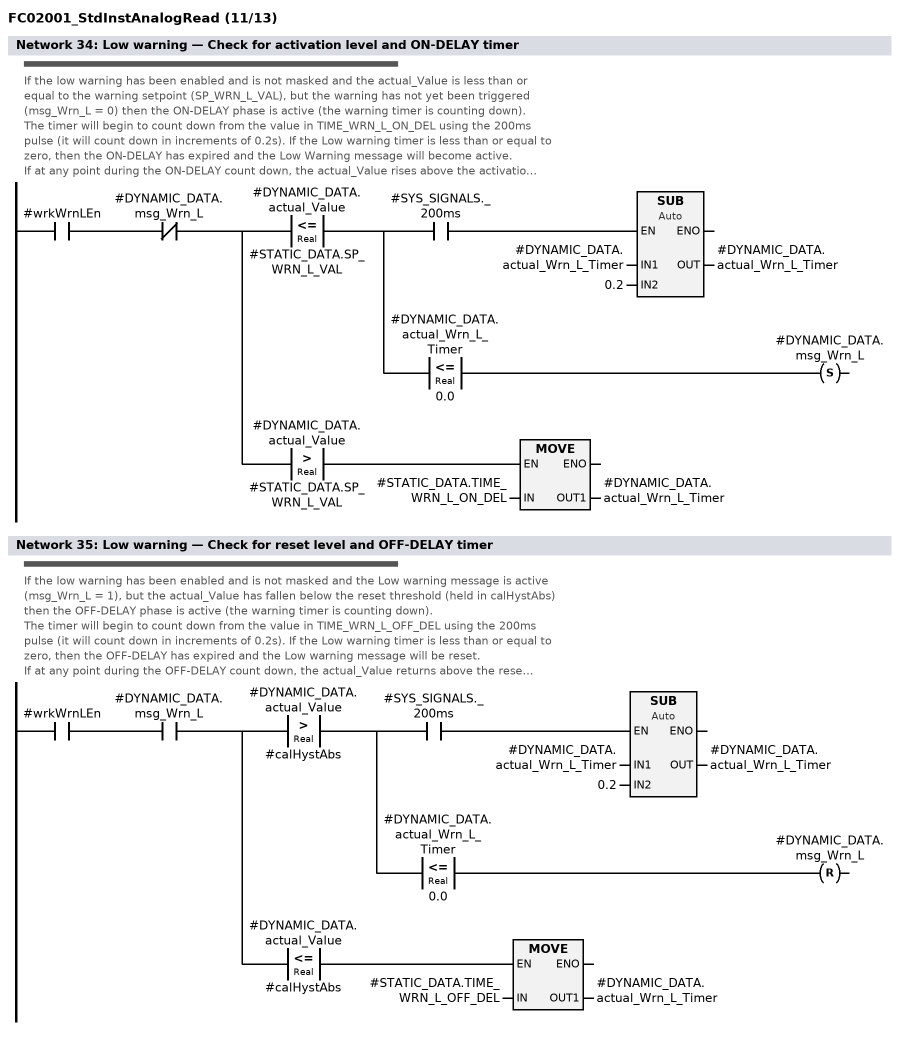
   RUNG wire#powerrail
      Contact( #wrkWrnLEn )
      I_Contact( #DYNAMIC_DATA.msg_Wrn_L )
      wire#w1
      { S7_Templates := "SrcType := Real" } LE_Contact(in1 := #DYNAMIC_DATA.actual_Value, in2 := #STATIC_DATA.SP_WRN_L_VAL)
      wire#w2
      Contact( #SYS_SIGNALS._200ms )
      Sub(in1 := #DYNAMIC_DATA.actual_Wrn_L_Timer, in2 := 0.2, out => #DYNAMIC_DATA.actual_Wrn_L_Timer)
   END_RUNG
   RUNG wire#w2
      { S7_Templates := "SrcType := Real" } LE_Contact(in1 := #DYNAMIC_DATA.actual_Wrn_L_Timer, in2 := 0.0)
      S_Coil( #DYNAMIC_DATA.msg_Wrn_L )
   END_RUNG
   RUNG wire#w1
      { S7_Templates := "SrcType := Real" } GT_Contact(in1 := #DYNAMIC_DATA.actual_Value, in2 := #STATIC_DATA.SP_WRN_L_VAL)
      { S7_GenerateENO := "TRUE" } Move(in := #STATIC_DATA.TIME_WRN_L_ON_DEL, out1 => #DYNAMIC_DATA.actual_Wrn_L_Timer)
   END_RUNG
   // the same network as SCL:
   #_w1 := #wrkWrnLEn AND NOT #DYNAMIC_DATA.msg_Wrn_L;
   #_w2 := #_w1 AND (#DYNAMIC_DATA.actual_Value <= #STATIC_DATA.SP_WRN_L_VAL);
   IF #_w2 AND #SYS_SIGNALS._200ms THEN
       #DYNAMIC_DATA.actual_Wrn_L_Timer := #DYNAMIC_DATA.actual_Wrn_L_Timer - 0.2;
   END_IF;
   IF #_w2 AND (#DYNAMIC_DATA.actual_Wrn_L_Timer <= 0.0) THEN #DYNAMIC_DATA.msg_Wrn_L := TRUE; END_IF;
   IF #_w1 AND (#DYNAMIC_DATA.actual_Value > #STATIC_DATA.SP_WRN_L_VAL) THEN
       #DYNAMIC_DATA.actual_Wrn_L_Timer := #STATIC_DATA.TIME_WRN_L_ON_DEL;
   END_IF;
END_REGION

REGION Network 35: Low warning — Check for reset level and OFF-DELAY timer
   // ▀▀▀▀▀▀▀▀▀▀▀▀▀▀▀▀▀▀▀▀▀▀▀▀▀▀▀▀▀▀▀▀▀▀▀▀▀▀▀▀▀▀▀▀
   // If the low warning has been enabled and is not masked and the Low warning message is active 
   // (msg_Wrn_L = 1), but the actual_Value has fallen below the reset threshold (held in calHystAbs) 
   // then the OFF-DELAY phase is active (the warning timer is counting down).
   // 
   // The timer will begin to count down from the value in TIME_WRN_L_OFF_DEL using the 200ms 
   // pulse (it will count down in increments of 0.2s). If the Low warning timer is less than or equal to 
   // zero, then the OFF-DELAY has expired and the Low warning message will be reset.
   // 
   // If at any point during the OFF-DELAY count down, the actual_Value returns above the reset
   // threshold (calHystAbs), the timer will be reset to the TIME_WRN_L_OFF_DEL value, forcing 
   // the OFF-DELAY to start again.
   // ▄▄▄▄▄▄▄▄▄▄▄▄▄▄▄▄▄▄▄▄▄▄▄▄▄▄▄▄▄▄▄▄▄▄▄▄▄▄▄▄▄▄▄▄
   RUNG wire#powerrail
      Contact( #wrkWrnLEn )
      Contact( #DYNAMIC_DATA.msg_Wrn_L )
      wire#w1
      { S7_Templates := "SrcType := Real" } GT_Contact(in1 := #DYNAMIC_DATA.actual_Value, in2 := #calHystAbs)
      wire#w2
      Contact( #SYS_SIGNALS._200ms )
      Sub(in1 := #DYNAMIC_DATA.actual_Wrn_L_Timer, in2 := 0.2, out => #DYNAMIC_DATA.actual_Wrn_L_Timer)
   END_RUNG
   RUNG wire#w2
      { S7_Templates := "SrcType := Real" } LE_Contact(in1 := #DYNAMIC_DATA.actual_Wrn_L_Timer, in2 := 0.0)
      R_Coil( #DYNAMIC_DATA.msg_Wrn_L )
   END_RUNG
   RUNG wire#w1
      { S7_Templates := "SrcType := Real" } LE_Contact(in1 := #DYNAMIC_DATA.actual_Value, in2 := #calHystAbs)
      { S7_GenerateENO := "TRUE" } Move(in := #STATIC_DATA.TIME_WRN_L_OFF_DEL, out1 => #DYNAMIC_DATA.actual_Wrn_L_Timer)
   END_RUNG
   // the same network as SCL:
   #_w1 := #wrkWrnLEn AND #DYNAMIC_DATA.msg_Wrn_L;
   #_w2 := #_w1 AND (#DYNAMIC_DATA.actual_Value > #calHystAbs);
   IF #_w2 AND #SYS_SIGNALS._200ms THEN
       #DYNAMIC_DATA.actual_Wrn_L_Timer := #DYNAMIC_DATA.actual_Wrn_L_Timer - 0.2;
   END_IF;
   IF #_w2 AND (#DYNAMIC_DATA.actual_Wrn_L_Timer <= 0.0) THEN #DYNAMIC_DATA.msg_Wrn_L := FALSE; END_IF;
   IF #_w1 AND (#DYNAMIC_DATA.actual_Value <= #calHystAbs) THEN
       #DYNAMIC_DATA.actual_Wrn_L_Timer := #STATIC_DATA.TIME_WRN_L_OFF_DEL;
   END_IF;
END_REGION

REGION Network 36: Status signals
   // ▀▀▀▀▀▀▀▀▀▀▀▀▀▀▀▀▀▀▀▀▀▀▀▀▀▀▀▀▀▀▀▀▀▀▀▀▀▀▀▀▀▀▀▀
   // The status signals for faults, alarms and warnings are either duplicates of the message signals 
   // (signals beginning with msg_) or logical combinations of them.
   // 
   // The following is a full list of the status signals:
   // 
   //  ――――――――――――――――――――――――――――――――――――――――――
   //  SIGNAL          FUNCTION            TYPE   DETAILS
   //  ――――――――――――――――――――――――――――――――――――――――――
   //  status_Alm_H       Identical to: msg_Alm_H    Bool    1 = high alm active, 0 = no alm
   // 
   //  status_Alm_L        Identical to: msg_Alm_L       Bool    1 = low alm active, 0 = no alm
   // 
   //  status_Wrn_H       Identical to: msg_Wrn_H    Bool    1 = high wrn active, 0 = no wrn
   // 
   //  status_Wrn_L        Identical to: msg_Wrn_L     Bool    1 = low wrn active, 0 = no wrn
   // 
   //  status_Alm_H_Mask     High alarm is masked        Bool    1 = alm masked, 0 = normal
   // 
   //  status_Alm_L_Mask      Low alarm is masked         Bool    1 = alm masked, 0 = normal
   // 
   //  status_Wrn_H_Mask     High warning is masked       Bool    1 = wrn masked, 0 = normal
   // 
   //  status_Wrn_L_Mask      Low warning is masked        Bool    1 = wrn masked, 0 = normal
   // 
   //  status_Alm_H_Dis         High alarm is disabled       Bool    1 = alm disabled, 0 = normal
   // 
   //  status_Alm_L_Dis          Low alarm is disabled        Bool    1 = alm disabled, 0 = normal
   // 
   //  status_Wrn_H_Dis         High warning is disabled   Bool    1 = wrn disabled, 0 = normal
   // 
   //  status_Wrn_L_Dis          Low warning is disabled       Bool    1 = wrn disabled, 0 = normal
   // 
   //  status_Fault      Indicates any of the msg_Flt    Bool    1 = fault active, 0 = healthy
   //                signals are active:
   //                  msg_Flt_UnderRange
   //                  msg_Flt_OverRange
   //                  msg_Flt_OutOfRange
   //                  msg_Flt_External 
   // 
   //                Note: msg_Flt_OutOfRange is already a combination of
   //                           msg_Flt_UnderRange and msg_Flt_OverRange
   // 
   //  status_SimOn      Status simulation mode on     Bool    1 = sim on, 0 = sim off
   // 
   //  status_RemoteOn     Status remote mode on     Bool    1 = rem on, 0 = rem off
   // 
   // 
   //  status_LocalOn      Status local mode on      Bool    1 = loc on, 0 = loc off 
   // 
   //  status_RLOff      Status ALL mode is on           Bool    1 = ALL mode on, 
   //                               0 = ALL mode off
   //  ――――――――――――――――――――――――――――――――――――――――――
   // ▄▄▄▄▄▄▄▄▄▄▄▄▄▄▄▄▄▄▄▄▄▄▄▄▄▄▄▄▄▄▄▄▄▄▄▄▄▄▄▄▄▄▄▄
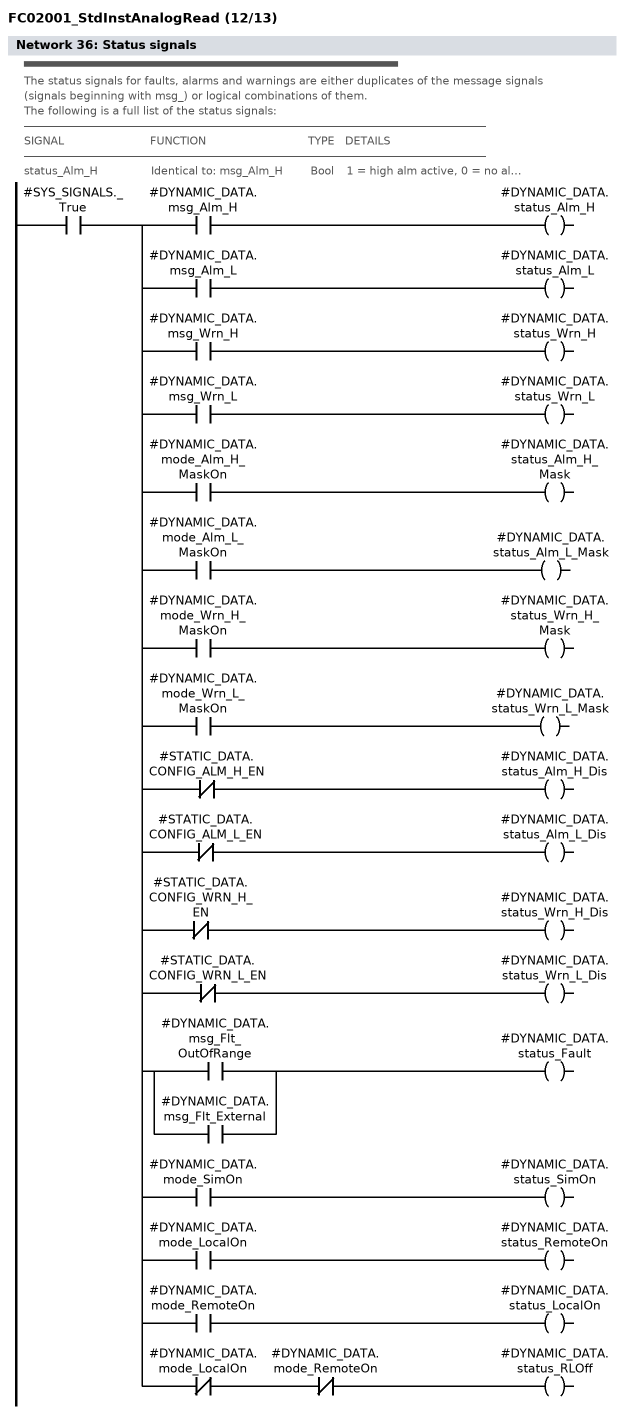
   RUNG wire#powerrail
      Contact( #SYS_SIGNALS._True )
      wire#w1
      Contact( #DYNAMIC_DATA.msg_Alm_H )
      Coil( #DYNAMIC_DATA.status_Alm_H )
   END_RUNG
   RUNG wire#w1
      Contact( #DYNAMIC_DATA.msg_Alm_L )
      Coil( #DYNAMIC_DATA.status_Alm_L )
   END_RUNG
   RUNG wire#w1
      Contact( #DYNAMIC_DATA.msg_Wrn_H )
      Coil( #DYNAMIC_DATA.status_Wrn_H )
   END_RUNG
   RUNG wire#w1
      Contact( #DYNAMIC_DATA.msg_Wrn_L )
      Coil( #DYNAMIC_DATA.status_Wrn_L )
   END_RUNG
   RUNG wire#w1
      Contact( #DYNAMIC_DATA.mode_Alm_H_MaskOn )
      Coil( #DYNAMIC_DATA.status_Alm_H_Mask )
   END_RUNG
   RUNG wire#w1
      Contact( #DYNAMIC_DATA.mode_Alm_L_MaskOn )
      Coil( #DYNAMIC_DATA.status_Alm_L_Mask )
   END_RUNG
   RUNG wire#w1
      Contact( #DYNAMIC_DATA.mode_Wrn_H_MaskOn )
      Coil( #DYNAMIC_DATA.status_Wrn_H_Mask )
   END_RUNG
   RUNG wire#w1
      Contact( #DYNAMIC_DATA.mode_Wrn_L_MaskOn )
      Coil( #DYNAMIC_DATA.status_Wrn_L_Mask )
   END_RUNG
   RUNG wire#w1
      I_Contact( #STATIC_DATA.CONFIG_ALM_H_EN )
      Coil( #DYNAMIC_DATA.status_Alm_H_Dis )
   END_RUNG
   RUNG wire#w1
      I_Contact( #STATIC_DATA.CONFIG_ALM_L_EN )
      Coil( #DYNAMIC_DATA.status_Alm_L_Dis )
   END_RUNG
   RUNG wire#w1
      I_Contact( #STATIC_DATA.CONFIG_WRN_H_EN )
      Coil( #DYNAMIC_DATA.status_Wrn_H_Dis )
   END_RUNG
   RUNG wire#w1
      I_Contact( #STATIC_DATA.CONFIG_WRN_L_EN )
      Coil( #DYNAMIC_DATA.status_Wrn_L_Dis )
   END_RUNG
   RUNG wire#w1
      Contact( #DYNAMIC_DATA.msg_Flt_OutOfRange )
      wire#w2
      Coil( #DYNAMIC_DATA.status_Fault )
   END_RUNG
   RUNG wire#w1
      Contact( #DYNAMIC_DATA.msg_Flt_External )
   END_RUNG wire#w2
   RUNG wire#w1
      Contact( #DYNAMIC_DATA.mode_SimOn )
      Coil( #DYNAMIC_DATA.status_SimOn )
   END_RUNG
   RUNG wire#w1
      Contact( #DYNAMIC_DATA.mode_LocalOn )
      Coil( #DYNAMIC_DATA.status_RemoteOn )
   END_RUNG
   RUNG wire#w1
      Contact( #DYNAMIC_DATA.mode_RemoteOn )
      Coil( #DYNAMIC_DATA.status_LocalOn )
   END_RUNG
   RUNG wire#w1
      I_Contact( #DYNAMIC_DATA.mode_LocalOn )
      I_Contact( #DYNAMIC_DATA.mode_RemoteOn )
      Coil( #DYNAMIC_DATA.status_RLOff )
   END_RUNG
   // the same network as SCL:
   #DYNAMIC_DATA.status_Alm_H := #SYS_SIGNALS._True AND #DYNAMIC_DATA.msg_Alm_H;
   #DYNAMIC_DATA.status_Alm_L := #SYS_SIGNALS._True AND #DYNAMIC_DATA.msg_Alm_L;
   #DYNAMIC_DATA.status_Wrn_H := #SYS_SIGNALS._True AND #DYNAMIC_DATA.msg_Wrn_H;
   #DYNAMIC_DATA.status_Wrn_L := #SYS_SIGNALS._True AND #DYNAMIC_DATA.msg_Wrn_L;
   #DYNAMIC_DATA.status_Alm_H_Mask := #SYS_SIGNALS._True AND #DYNAMIC_DATA.mode_Alm_H_MaskOn;
   #DYNAMIC_DATA.status_Alm_L_Mask := #SYS_SIGNALS._True AND #DYNAMIC_DATA.mode_Alm_L_MaskOn;
   #DYNAMIC_DATA.status_Wrn_H_Mask := #SYS_SIGNALS._True AND #DYNAMIC_DATA.mode_Wrn_H_MaskOn;
   #DYNAMIC_DATA.status_Wrn_L_Mask := #SYS_SIGNALS._True AND #DYNAMIC_DATA.mode_Wrn_L_MaskOn;
   #DYNAMIC_DATA.status_Alm_H_Dis := #SYS_SIGNALS._True AND NOT #STATIC_DATA.CONFIG_ALM_H_EN;
   #DYNAMIC_DATA.status_Alm_L_Dis := #SYS_SIGNALS._True AND NOT #STATIC_DATA.CONFIG_ALM_L_EN;
   #DYNAMIC_DATA.status_Wrn_H_Dis := #SYS_SIGNALS._True AND NOT #STATIC_DATA.CONFIG_WRN_H_EN;
   #DYNAMIC_DATA.status_Wrn_L_Dis := #SYS_SIGNALS._True AND NOT #STATIC_DATA.CONFIG_WRN_L_EN;
   #DYNAMIC_DATA.status_Fault := #SYS_SIGNALS._True AND (#DYNAMIC_DATA.msg_Flt_OutOfRange OR #DYNAMIC_DATA.msg_Flt_External);
   #DYNAMIC_DATA.status_SimOn := #SYS_SIGNALS._True AND #DYNAMIC_DATA.mode_SimOn;
   #DYNAMIC_DATA.status_RemoteOn := #SYS_SIGNALS._True AND #DYNAMIC_DATA.mode_LocalOn;
   #DYNAMIC_DATA.status_LocalOn := #SYS_SIGNALS._True AND #DYNAMIC_DATA.mode_RemoteOn;
   #DYNAMIC_DATA.status_RLOff := #SYS_SIGNALS._True AND NOT #DYNAMIC_DATA.mode_LocalOn AND NOT #DYNAMIC_DATA.mode_RemoteOn;
END_REGION

REGION Network 37: LICENCE AND CONTACT INFORMATION
   // ▀▀▀▀▀▀▀▀▀▀▀▀▀▀▀▀▀▀▀▀▀▀▀▀▀▀▀▀▀▀▀▀▀▀▀▀▀▀▀▀▀▀▀▀
   // LICENCE AND CONTACT INFORMATION
   // 
   // This software and its associated documentation is made available under the MIT Licence:
   // 
   // ════════════════════════════════════════════
   // 
   // The MIT License (MIT)
   // 
   // Copyright © 2020 Michael Gledhill
   // 
   // Permission is hereby granted, free of charge, to any person obtaining a copy of this software 
   // and associated documentation files (the “Software”), to deal in the Software without restriction, 
   // including without limitation the rights to use, copy, modify, merge, publish, distribute, 
   // sublicense, and/or sell copies of the Software, and to permit persons to whom the Software is 
   // furnished to do so, subject to the following conditions: 
   // 
   // The above copyright notice and this permission notice shall be included in all copies or 
   // substantial portions of the Software.
   // 
   // THE SOFTWARE IS PROVIDED “AS IS”, WITHOUT WARRANTY OF ANY KIND, EXPRESS OR IMPLIED, 
   // INCLUDING BUT NOT LIMITED TO THE WARRANTIES OF MERCHANTABILITY, FITNESS FOR A 
   // PARTICULAR PURPOSE AND NON-INFRINGEMENT. IN NO EVENT SHALL THE AUTHORS OR COPYRIGHT 
   // HOLDERS BE LIABLE FOR ANY CLAIM, DAMAGES OR OTHER LIABILITY, WHETHER IN AN ACTION OF 
   // CONTRACT, TORT OR OTHERWISE, ARISING FROM, OUT OF OR IN CONNECTION WITH THE SOFTWARE 
   // OR THE USE OR OTHER DEALINGS IN THE SOFTWARE.
   // 
   // ════════════════════════════════════════════
   //                    ┌────────────┐
   // You can reach the author by email here:   │  mg@practicalseries.com  │
   //                    └────────────┘
   // Questions, corrections, constructive criticism and complaints (polite ones) are invited.
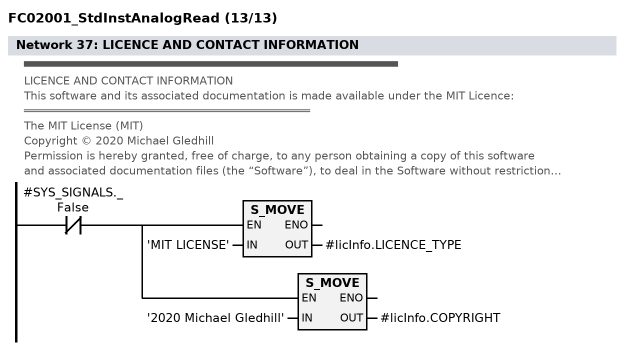
   RUNG wire#powerrail
      I_Contact( #SYS_SIGNALS._False )
      wire#w1
      S_Move(in := 'MIT LICENSE', out => #licInfo.LICENCE_TYPE)
   END_RUNG
   RUNG wire#w1
      S_Move(in := '2020 Michael Gledhill', out => #licInfo.COPYRIGHT)
   END_RUNG
   // the same network as SCL:
   IF NOT #SYS_SIGNALS._False THEN
       #licInfo.LICENCE_TYPE := 'MIT LICENSE';
       #licInfo.COPYRIGHT := '2020 Michael Gledhill';
   END_IF;
END_REGION
END_FUNCTION
